LIN {X 0,Y 541.517,Z 483.658,A -85,B 0,C 180,E1 4032.092,E2 4032.092} C_VEL
LIN {X 0,Y 540.4,Z 508.601,A -85,B 0,C 180,E1 4034.781,E2 4034.781} C_VEL
LIN {X 0,Y 539.621,Z 531.792,A -85,B 0,C 180,E1 4038.266,E2 4038.266} C_VEL
LIN {X 0,Y 539.263,Z 546.74,A -85,B 0,C 180,E1 4041.527,E2 4041.527} C_VEL
LIN {X 0,Y 539.076,Z 557.16,A -85,B 0,C 180,E1 4045.169,E2 4045.169} C_VEL
LIN {X 0,Y 538.968,Z 561.446,A -85,B 0,C 180,E1 4048.393,E2 4048.393} C_VEL
LIN {X 0,Y 538.979,Z 561.385,A -85,B 0,C 180,E1 4051.612,E2 4051.612} C_VEL
LIN {X 0,Y 539.098,Z 556.976,A -85,B 0,C 180,E1 4054.835,E2 4054.835} C_VEL
LIN {X 0,Y 539.274,Z 546.384,A -85,B 0,C 180,E1 4058.478,E2 4058.478} C_VEL
LIN {X 0,Y 539.639,Z 530.084,A -85,B 0,C 180,E1 4061.943,E2 4061.943} C_VEL
LIN {X 0,Y 540.473,Z 506.897,A -85,B 0,C 180,E1 4065.337,E2 4065.337} C_VEL
LIN {X 0,Y 541.656,Z 481.261,A -85,B 0,C 180,E1 4068.039,E2 4068.039} C_VEL
LIN {X 0,Y 543.03,Z 451.784,A -85,B 0,C 180,E1 4070.227,E2 4070.227} C_VEL
LIN {X 0,Y 544.237,Z 421.039,A -85,B 0,C 180,E1 4071.776,E2 4071.776} C_VEL
LIN {X 0,Y 544.348,Z 387.144,A -85,B 0,C 180,E1 4072.819,E2 4072.819} C_VEL
LIN {X 0,Y 538.422,Z 370.16,A -85,B 0,C 180,E1 4073.523,E2 4073.523} C_VEL
LIN {X 0,Y 538.216,Z 370.16,A -85,B 0,C 180,E1 4079.313,E2 4079.313} C_VEL
LIN {X 0,Y 538.135,Z 370.16,A -85,B 0,C 180,E1 4085.331,E2 4085.331} C_VEL
LIN {X 0,Y 538.098,Z 370.16,A -85,B 0,C 180,E1 4090.57,E2 4090.57} C_VEL
LIN {X 0,Y 538.199,Z 370.16,A -85,B 0,C 180,E1 4097.005,E2 4097.005} C_VEL
LIN {X 0,Y 538.211,Z 370.16,A -85,B 0,C 180,E1 4101.967,E2 4101.967} C_VEL
LIN {X 0,Y 538.141,Z 370.16,A -85,B 0,C 180,E1 4107.691,E2 4107.691} C_VEL
LIN {X 0,Y 538.372,Z 370.16,A -85,B 0,C 180,E1 4113.263,E2 4113.263} C_VEL
LIN {X 0,Y 538.444,Z 370.16,A -85,B 0,C 180,E1 4118.562,E2 4118.562} C_VEL
LIN {X 0,Y 538.537,Z 370.16,A -85,B 0,C 180,E1 4123.674,E2 4123.674} C_VEL
LIN {X 0,Y 538.543,Z 370.16,A -85,B 0,C 180,E1 4128.652,E2 4128.652} C_VEL
LIN {X 0,Y 538.567,Z 370.16,A -85,B 0,C 180,E1 4133.545,E2 4133.545} C_VEL
LIN {X 0,Y 538.637,Z 370.16,A -85,B 0,C 180,E1 4138.39,E2 4138.39} C_VEL
LIN {X 0,Y 538.602,Z 370.16,A -85,B 0,C 180,E1 4143.224,E2 4143.224} C_VEL
LIN {X 0,Y 538.512,Z 370.16,A -85,B 0,C 180,E1 4148.082,E2 4148.082} C_VEL
LIN {X 0,Y 538.484,Z 370.16,A -85,B 0,C 180,E1 4152.999,E2 4152.999} C_VEL
LIN {X 0,Y 538.425,Z 370.16,A -85,B 0,C 180,E1 4158.018,E2 4158.018} C_VEL
LIN {X 0,Y 538.392,Z 370.16,A -85,B 0,C 180,E1 4163.184,E2 4163.184} C_VEL
LIN {X 0,Y 538.361,Z 370.16,A -85,B 0,C 180,E1 4165.152,E2 4165.152} C_VEL
LIN {X 0,Y 537.043,Z 370.16,A -85,B 0,C 180,E1 4166.074,E2 4166.074} C_VEL
LIN {X 0,Y 530.382,Z 370.16,A -85,B 0,C 180,E1 4168.584,E2 4168.584} C_VEL
LIN {X 0,Y 530.303,Z 370.16,A -85,B 0,C 180,E1 4168.822,E2 4168.822} C_VEL
LIN {X 0,Y 530.316,Z 370.16,A -85,B 0,C 180,E1 4174.817,E2 4174.817} C_VEL
LIN {X 0,Y 530.257,Z 370.16,A -85,B 0,C 180,E1 4181.047,E2 4181.047} C_VEL
LIN {X 0,Y 530.306,Z 370.16,A -85,B 0,C 180,E1 4186.749,E2 4186.749} C_VEL
LIN {X 0,Y 530.279,Z 370.16,A -85,B 0,C 180,E1 4193.16,E2 4193.16} C_VEL
LIN {X 0,Y 530.257,Z 370.16,A -85,B 0,C 180,E1 4199.072,E2 4199.072} C_VEL
LIN {X 0,Y 530.443,Z 370.823,A -85,B 0,C 180,E1 4200.434,E2 4200.434} C_VEL
LIN {X 0,Y 539.972,Z 394.145,A -85,B 0,C 180,E1 4201.321,E2 4201.321} C_VEL
LIN {X 0,Y 539.426,Z 441.23,A -85,B 0,C 180,E1 4202.159,E2 4202.159} C_VEL
LIN {X 0,Y 538.185,Z 477.288,A -85,B 0,C 180,E1 4203.418,E2 4203.418} C_VEL
LIN {X 0,Y 536.636,Z 511.971,A -85,B 0,C 180,E1 4205.296,E2 4205.296} C_VEL
LIN {X 0,Y 534.86,Z 545.508,A -85,B 0,C 180,E1 4207.882,E2 4207.882} C_VEL
LIN {X 0,Y 533.35,Z 574.49,A -85,B 0,C 180,E1 4210.945,E2 4210.945} C_VEL
LIN {X 0,Y 532.266,Z 598.279,A -85,B 0,C 180,E1 4214.321,E2 4214.321} C_VEL
LIN {X 0,Y 531.508,Z 617.476,A -85,B 0,C 180,E1 4218.08,E2 4218.08} C_VEL
LIN {X 0,Y 531.215,Z 630.601,A -85,B 0,C 180,E1 4221.805,E2 4221.805} C_VEL
LIN {X 0,Y 531.108,Z 637.962,A -85,B 0,C 180,E1 4225.092,E2 4225.092} C_VEL
LIN {X 0,Y 531.031,Z 641.508,A -85,B 0,C 180,E1 4228.364,E2 4228.364} C_VEL
LIN {X 0,Y 531.091,Z 641.512,A -85,B 0,C 180,E1 4231.631,E2 4231.631} C_VEL
LIN {X 0,Y 531.113,Z 637.97,A -85,B 0,C 180,E1 4234.903,E2 4234.903} C_VEL
LIN {X 0,Y 531.284,Z 628.183,A -85,B 0,C 180,E1 4239.014,E2 4239.014} C_VEL
LIN {X 0,Y 531.626,Z 613.791,A -85,B 0,C 180,E1 4242.748,E2 4242.748} C_VEL
LIN {X 0,Y 532.369,Z 594.338,A -85,B 0,C 180,E1 4246.307,E2 4246.307} C_VEL
LIN {X 0,Y 533.592,Z 569.267,A -85,B 0,C 180,E1 4249.687,E2 4249.687} C_VEL
LIN {X 0,Y 535.172,Z 539.83,A -85,B 0,C 180,E1 4252.617,E2 4252.617} C_VEL
LIN {X 0,Y 536.928,Z 506.945,A -85,B 0,C 180,E1 4255.018,E2 4255.018} C_VEL
LIN {X 0,Y 538.474,Z 472.313,A -85,B 0,C 180,E1 4256.797,E2 4256.797} C_VEL
LIN {X 0,Y 539.646,Z 435.196,A -85,B 0,C 180,E1 4257.986,E2 4257.986} C_VEL
LIN {X 0,Y 539.599,Z 392.517,A -85,B 0,C 180,E1 4258.725,E2 4258.725} C_VEL
LIN {X 0,Y 530.512,Z 370.16,A -85,B 0,C 180,E1 4259.603,E2 4259.603} C_VEL
LIN {X 0,Y 530.417,Z 370.16,A -85,B 0,C 180,E1 4264.806,E2 4264.806} C_VEL
LIN {X 0,Y 530.215,Z 370.16,A -85,B 0,C 180,E1 4271.047,E2 4271.047} C_VEL
LIN {X 0,Y 530.123,Z 370.16,A -85,B 0,C 180,E1 4276.733,E2 4276.733} C_VEL
LIN {X 0,Y 530.197,Z 370.16,A -85,B 0,C 180,E1 4283.155,E2 4283.155} C_VEL
LIN {X 0,Y 530.295,Z 370.16,A -85,B 0,C 180,E1 4289.077,E2 4289.077} C_VEL
LIN {X 0,Y 530.5,Z 370.16,A -85,B 0,C 180,E1 4294.654,E2 4294.654} C_VEL
LIN {X 0,Y 530.61,Z 370.872,A -85,B 0,C 180,E1 4296.73,E2 4296.73} C_VEL
LIN {X 0,Y 536.183,Z 392.946,A -85,B 0,C 180,E1 4297.301,E2 4297.301} C_VEL
LIN {X 0,Y 535.619,Z 427.462,A -85,B 0,C 180,E1 4298.388,E2 4298.388} C_VEL
LIN {X 0,Y 534.637,Z 459.023,A -85,B 0,C 180,E1 4300.06,E2 4300.06} C_VEL
LIN {X 0,Y 533.537,Z 487.309,A -85,B 0,C 180,E1 4302.269,E2 4302.269} C_VEL
LIN {X 0,Y 532.555,Z 511.968,A -85,B 0,C 180,E1 4304.986,E2 4304.986} C_VEL
LIN {X 0,Y 531.776,Z 531.931,A -85,B 0,C 180,E1 4308.087,E2 4308.087} C_VEL
LIN {X 0,Y 531.321,Z 548.213,A -85,B 0,C 180,E1 4311.808,E2 4311.808} C_VEL
LIN {X 0,Y 531.198,Z 557.105,A -85,B 0,C 180,E1 4315.094,E2 4315.094} C_VEL
LIN {X 0,Y 531.08,Z 561.45,A -85,B 0,C 180,E1 4318.365,E2 4318.365} C_VEL
LIN {X 0,Y 531.044,Z 561.418,A -85,B 0,C 180,E1 4321.633,E2 4321.633} C_VEL
LIN {X 0,Y 531.185,Z 556.932,A -85,B 0,C 180,E1 4324.904,E2 4324.904} C_VEL
LIN {X 0,Y 531.399,Z 546.438,A -85,B 0,C 180,E1 4328.601,E2 4328.601} C_VEL
LIN {X 0,Y 531.839,Z 529.134,A -85,B 0,C 180,E1 4332.326,E2 4332.326} C_VEL
LIN {X 0,Y 532.702,Z 507.725,A -85,B 0,C 180,E1 4335.45,E2 4335.45} C_VEL
LIN {X 0,Y 533.755,Z 482.611,A -85,B 0,C 180,E1 4338.067,E2 4338.067} C_VEL
LIN {X 0,Y 534.91,Z 453.057,A -85,B 0,C 180,E1 4340.248,E2 4340.248} C_VEL
LIN {X 0,Y 535.928,Z 420.413,A -85,B 0,C 180,E1 4341.854,E2 4341.854} C_VEL
LIN {X 0,Y 535.687,Z 387.806,A -85,B 0,C 180,E1 4342.835,E2 4342.835} C_VEL
LIN {X 0,Y 530.468,Z 370.16,A -85,B 0,C 180,E1 4343.4,E2 4343.4} C_VEL
LIN {X 0,Y 530.383,Z 370.16,A -85,B 0,C 180,E1 4349.027,E2 4349.027} C_VEL
LIN {X 0,Y 530.341,Z 370.16,A -85,B 0,C 180,E1 4354.813,E2 4354.813} C_VEL
LIN {X 0,Y 530.263,Z 370.16,A -85,B 0,C 180,E1 4361.044,E2 4361.044} C_VEL
LIN {X 0,Y 530.33,Z 370.16,A -85,B 0,C 180,E1 4366.758,E2 4366.758} C_VEL
LIN {X 0,Y 530.275,Z 370.16,A -85,B 0,C 180,E1 4373.166,E2 4373.166} C_VEL
LIN {X 0,Y 530.286,Z 370.16,A -85,B 0,C 180,E1 4379.08,E2 4379.08} C_VEL
LIN {X 0,Y 530.494,Z 370.16,A -85,B 0,C 180,E1 4384.657,E2 4384.657} C_VEL
LIN {X 0,Y 530.579,Z 370.16,A -85,B 0,C 180,E1 4385.986,E2 4385.986} C_VEL
LIN {X 0,Y 537.911,Z 392.099,A -85,B 0,C 180,E1 4386.837,E2 4386.837} C_VEL
LIN {X 0,Y 537.063,Z 426.025,A -85,B 0,C 180,E1 4387.945,E2 4387.945} C_VEL
LIN {X 0,Y 535.666,Z 456.498,A -85,B 0,C 180,E1 4389.59,E2 4389.59} C_VEL
LIN {X 0,Y 534.104,Z 484.887,A -85,B 0,C 180,E1 4391.835,E2 4391.835} C_VEL
LIN {X 0,Y 532.815,Z 509.576,A -85,B 0,C 180,E1 4394.554,E2 4394.554} C_VEL
LIN {X 0,Y 531.861,Z 529.926,A -85,B 0,C 180,E1 4397.676,E2 4397.676} C_VEL
LIN {X 0,Y 531.395,Z 546.737,A -85,B 0,C 180,E1 4401.4,E2 4401.4} C_VEL
LIN {X 0,Y 531.186,Z 557.158,A -85,B 0,C 180,E1 4405.098,E2 4405.098} C_VEL
LIN {X 0,Y 531.065,Z 561.445,A -85,B 0,C 180,E1 4408.369,E2 4408.369} C_VEL
LIN {X 0,Y 531.076,Z 561.385,A -85,B 0,C 180,E1 4411.636,E2 4411.636} C_VEL
LIN {X 0,Y 531.207,Z 556.977,A -85,B 0,C 180,E1 4414.907,E2 4414.907} C_VEL
LIN {X 0,Y 531.404,Z 546.387,A -85,B 0,C 180,E1 4418.604,E2 4418.604} C_VEL
LIN {X 0,Y 531.909,Z 529.402,A -85,B 0,C 180,E1 4422.328,E2 4422.328} C_VEL
LIN {X 0,Y 532.871,Z 509.001,A -85,B 0,C 180,E1 4425.428,E2 4425.428} C_VEL
LIN {X 0,Y 534.174,Z 483.9,A -85,B 0,C 180,E1 4428.168,E2 4428.168} C_VEL
LIN {X 0,Y 535.714,Z 454.866,A -85,B 0,C 180,E1 4430.426,E2 4430.426} C_VEL
LIN {X 0,Y 537.128,Z 423.446,A -85,B 0,C 180,E1 4432.08,E2 4432.08} C_VEL
LIN {X 0,Y 537.394,Z 389.167,A -85,B 0,C 180,E1 4433.17,E2 4433.17} C_VEL
LIN {X 0,Y 530.53,Z 370.16,A -85,B 0,C 180,E1 4433.979,E2 4433.979} C_VEL
LIN {X 0,Y 530.324,Z 370.16,A -85,B 0,C 180,E1 4439.035,E2 4439.035} C_VEL
LIN {X 0,Y 530.253,Z 370.16,A -85,B 0,C 180,E1 4444.824,E2 4444.824} C_VEL
LIN {X 0,Y 530.155,Z 370.16,A -85,B 0,C 180,E1 4451.059,E2 4451.059} C_VEL
LIN {X 0,Y 530.295,Z 370.16,A -85,B 0,C 180,E1 4456.753,E2 4456.753} C_VEL
LIN {X 0,Y 530.218,Z 370.16,A -85,B 0,C 180,E1 4463.085,E2 4463.085} C_VEL
LIN {X 0,Y 530.24,Z 370.16,A -85,B 0,C 180,E1 4469.076,E2 4469.076} C_VEL
LIN {X 0,Y 530.498,Z 370.16,A -85,B 0,C 180,E1 4474.657,E2 4474.657} C_VEL
LIN {X 0,Y 530.632,Z 370.16,A -85,B 0,C 180,E1 4480.314,E2 4480.314} C_VEL
LIN {X 0,Y 530.693,Z 370.16,A -85,B 0,C 180,E1 4485.924,E2 4485.924} C_VEL
LIN {X 0,Y 530.722,Z 370.16,A -85,B 0,C 180,E1 4491.801,E2 4491.801} C_VEL
LIN {X 0,Y 530.88,Z 370.16,A -85,B 0,C 180,E1 4496.732,E2 4496.732} C_VEL
LIN {X 0,Y 530.952,Z 370.16,A -85,B 0,C 180,E1 4501.635,E2 4501.635} C_VEL
LIN {X 0,Y 530.841,Z 370.16,A -85,B 0,C 180,E1 4506.551,E2 4506.551} C_VEL
LIN {X 0,Y 530.652,Z 370.16,A -85,B 0,C 180,E1 4511.521,E2 4511.521} C_VEL
LIN {X 0,Y 530.549,Z 370.16,A -85,B 0,C 180,E1 4516.581,E2 4516.581} C_VEL
LIN {X 0,Y 530.524,Z 370.16,A -85,B 0,C 180,E1 4521.777,E2 4521.777} C_VEL
LIN {X 0,Y 530.327,Z 370.16,A -85,B 0,C 180,E1 4527.748,E2 4527.748} C_VEL
LIN {X 0,Y 530.303,Z 370.16,A -85,B 0,C 180,E1 4528.822,E2 4528.822} C_VEL
LIN {X 0,Y 527.774,Z 370.16,A -85,B 0,C 180,E1 4530.211,E2 4530.211} C_VEL
LIN {X 0,Y 522.404,Z 370.16,A -85,B 0,C 180,E1 4532.292,E2 4532.292} C_VEL
LIN {X 0,Y 522.331,Z 370.16,A -85,B 0,C 180,E1 4532.533,E2 4532.533} C_VEL
LIN {X 0,Y 522.368,Z 370.16,A -85,B 0,C 180,E1 4538.505,E2 4538.505} C_VEL
LIN {X 0,Y 522.34,Z 370.16,A -85,B 0,C 180,E1 4544.076,E2 4544.076} C_VEL
LIN {X 0,Y 522.375,Z 370.16,A -85,B 0,C 180,E1 4550.384,E2 4550.384} C_VEL
LIN {X 0,Y 522.337,Z 370.16,A -85,B 0,C 180,E1 4556.583,E2 4556.583} C_VEL
LIN {X 0,Y 522.483,Z 370.16,A -85,B 0,C 180,E1 4559.982,E2 4559.982} C_VEL
LIN {X 0,Y 533.184,Z 398.599,A -85,B 0,C 180,E1 4560.988,E2 4560.988} C_VEL
LIN {X 0,Y 532.347,Z 444.004,A -85,B 0,C 180,E1 4561.837,E2 4561.837} C_VEL
LIN {X 0,Y 530.986,Z 479.733,A -85,B 0,C 180,E1 4563.144,E2 4563.144} C_VEL
LIN {X 0,Y 529.159,Z 515.25,A -85,B 0,C 180,E1 4565.149,E2 4565.149} C_VEL
LIN {X 0,Y 527.308,Z 546.909,A -85,B 0,C 180,E1 4567.684,E2 4567.684} C_VEL
LIN {X 0,Y 525.751,Z 574.49,A -85,B 0,C 180,E1 4570.659,E2 4570.659} C_VEL
LIN {X 0,Y 524.481,Z 598.279,A -85,B 0,C 180,E1 4574.082,E2 4574.082} C_VEL
LIN {X 0,Y 523.667,Z 617.477,A -85,B 0,C 180,E1 4577.899,E2 4577.899} C_VEL
LIN {X 0,Y 523.335,Z 630.601,A -85,B 0,C 180,E1 4581.681,E2 4581.681} C_VEL
LIN {X 0,Y 523.213,Z 637.961,A -85,B 0,C 180,E1 4585.018,E2 4585.018} C_VEL
LIN {X 0,Y 523.146,Z 641.509,A -85,B 0,C 180,E1 4588.339,E2 4588.339} C_VEL
LIN {X 0,Y 523.202,Z 641.512,A -85,B 0,C 180,E1 4591.656,E2 4591.656} C_VEL
LIN {X 0,Y 523.207,Z 637.97,A -85,B 0,C 180,E1 4594.977,E2 4594.977} C_VEL
LIN {X 0,Y 523.387,Z 629.464,A -85,B 0,C 180,E1 4598.732,E2 4598.732} C_VEL
LIN {X 0,Y 523.756,Z 615.735,A -85,B 0,C 180,E1 4602.518,E2 4602.518} C_VEL
LIN {X 0,Y 524.554,Z 595.663,A -85,B 0,C 180,E1 4606.341,E2 4606.341} C_VEL
LIN {X 0,Y 525.905,Z 571.028,A -85,B 0,C 180,E1 4609.768,E2 4609.768} C_VEL
LIN {X 0,Y 527.674,Z 541.222,A -85,B 0,C 180,E1 4612.834,E2 4612.834} C_VEL
LIN {X 0,Y 529.587,Z 508.646,A -85,B 0,C 180,E1 4615.276,E2 4615.276} C_VEL
LIN {X 0,Y 531.303,Z 473.736,A -85,B 0,C 180,E1 4617.121,E2 4617.121} C_VEL
LIN {X 0,Y 532.619,Z 437.259,A -85,B 0,C 180,E1 4618.34,E2 4618.34} C_VEL
LIN {X 0,Y 532.484,Z 394.319,A -85,B 0,C 180,E1 4619.117,E2 4619.117} C_VEL
LIN {X 0,Y 522.573,Z 370.16,A -85,B 0,C 180,E1 4620.064,E2 4620.064} C_VEL
LIN {X 0,Y 522.407,Z 370.16,A -85,B 0,C 180,E1 4625.763,E2 4625.763} C_VEL
LIN {X 0,Y 522.275,Z 370.16,A -85,B 0,C 180,E1 4631.81,E2 4631.81} C_VEL
LIN {X 0,Y 522.231,Z 370.16,A -85,B 0,C 180,E1 4638.182,E2 4638.182} C_VEL
LIN {X 0,Y 522.261,Z 370.16,A -85,B 0,C 180,E1 4644.566,E2 4644.566} C_VEL
LIN {X 0,Y 522.4,Z 370.16,A -85,B 0,C 180,E1 4650.483,E2 4650.483} C_VEL
LIN {X 0,Y 522.638,Z 370.16,A -85,B 0,C 180,E1 4656.388,E2 4656.388} C_VEL
LIN {X 0,Y 528.676,Z 392.668,A -85,B 0,C 180,E1 4657.022,E2 4657.022} C_VEL
LIN {X 0,Y 528.103,Z 427.602,A -85,B 0,C 180,E1 4658.119,E2 4658.119} C_VEL
LIN {X 0,Y 527.054,Z 459.805,A -85,B 0,C 180,E1 4659.836,E2 4659.836} C_VEL
LIN {X 0,Y 525.853,Z 488.687,A -85,B 0,C 180,E1 4662.127,E2 4662.127} C_VEL
LIN {X 0,Y 524.81,Z 513.709,A -85,B 0,C 180,E1 4664.951,E2 4664.951} C_VEL
LIN {X 0,Y 523.97,Z 533.559,A -85,B 0,C 180,E1 4668.119,E2 4668.119} C_VEL
LIN {X 0,Y 523.494,Z 548.685,A -85,B 0,C 180,E1 4671.685,E2 4671.685} C_VEL
LIN {X 0,Y 523.3,Z 557.335,A -85,B 0,C 180,E1 4675.02,E2 4675.02} C_VEL
LIN {X 0,Y 523.192,Z 561.543,A -85,B 0,C 180,E1 4678.341,E2 4678.341} C_VEL
LIN {X 0,Y 523.157,Z 561.506,A -85,B 0,C 180,E1 4681.657,E2 4681.657} C_VEL
LIN {X 0,Y 523.292,Z 557.138,A -85,B 0,C 180,E1 4684.978,E2 4684.978} C_VEL
LIN {X 0,Y 523.55,Z 546.828,A -85,B 0,C 180,E1 4688.731,E2 4688.731} C_VEL
LIN {X 0,Y 524.017,Z 530.672,A -85,B 0,C 180,E1 4692.301,E2 4692.301} C_VEL
LIN {X 0,Y 524.957,Z 509.65,A -85,B 0,C 180,E1 4695.47,E2 4695.47} C_VEL
LIN {X 0,Y 526.07,Z 484.343,A -85,B 0,C 180,E1 4698.188,E2 4698.188} C_VEL
LIN {X 0,Y 527.33,Z 454.86,A -85,B 0,C 180,E1 4700.42,E2 4700.42} C_VEL
LIN {X 0,Y 528.401,Z 423.505,A -85,B 0,C 180,E1 4702.028,E2 4702.028} C_VEL
LIN {X 0,Y 528.546,Z 390.358,A -85,B 0,C 180,E1 4703.074,E2 4703.074} C_VEL
LIN {X 0,Y 522.542,Z 370.16,A -85,B 0,C 180,E1 4703.69,E2 4703.69} C_VEL
LIN {X 0,Y 522.406,Z 370.16,A -85,B 0,C 180,E1 4709.616,E2 4709.616} C_VEL
LIN {X 0,Y 522.391,Z 370.16,A -85,B 0,C 180,E1 4715.765,E2 4715.765} C_VEL
LIN {X 0,Y 522.352,Z 370.16,A -85,B 0,C 180,E1 4721.803,E2 4721.803} C_VEL
LIN {X 0,Y 522.397,Z 370.16,A -85,B 0,C 180,E1 4728.202,E2 4728.202} C_VEL
LIN {X 0,Y 522.309,Z 370.16,A -85,B 0,C 180,E1 4734.573,E2 4734.573} C_VEL
LIN {X 0,Y 522.392,Z 370.16,A -85,B 0,C 180,E1 4740.486,E2 4740.486} C_VEL
LIN {X 0,Y 522.624,Z 370.16,A -85,B 0,C 180,E1 4745.523,E2 4745.523} C_VEL
LIN {X 0,Y 530.956,Z 394.225,A -85,B 0,C 180,E1 4746.475,E2 4746.475} C_VEL
LIN {X 0,Y 529.995,Z 427.507,A -85,B 0,C 180,E1 4747.602,E2 4747.602} C_VEL
LIN {X 0,Y 528.398,Z 458.785,A -85,B 0,C 180,E1 4749.337,E2 4749.337} C_VEL
LIN {X 0,Y 526.663,Z 487.353,A -85,B 0,C 180,E1 4751.682,E2 4751.682} C_VEL
LIN {X 0,Y 525.148,Z 512.132,A -85,B 0,C 180,E1 4754.537,E2 4754.537} C_VEL
LIN {X 0,Y 524.103,Z 533.026,A -85,B 0,C 180,E1 4757.914,E2 4757.914} C_VEL
LIN {X 0,Y 523.566,Z 547.353,A -85,B 0,C 180,E1 4761.271,E2 4761.271} C_VEL
LIN {X 0,Y 523.287,Z 557.383,A -85,B 0,C 180,E1 4765.023,E2 4765.023} C_VEL
LIN {X 0,Y 523.177,Z 561.528,A -85,B 0,C 180,E1 4768.344,E2 4768.344} C_VEL
LIN {X 0,Y 523.189,Z 561.47,A -85,B 0,C 180,E1 4771.661,E2 4771.661} C_VEL
LIN {X 0,Y 523.314,Z 557.211,A -85,B 0,C 180,E1 4774.981,E2 4774.981} C_VEL
LIN {X 0,Y 523.595,Z 547.027,A -85,B 0,C 180,E1 4778.734,E2 4778.734} C_VEL
LIN {X 0,Y 524.163,Z 531.432,A -85,B 0,C 180,E1 4782.301,E2 4782.301} C_VEL
LIN {X 0,Y 525.324,Z 509.902,A -85,B 0,C 180,E1 4785.677,E2 4785.677} C_VEL
LIN {X 0,Y 526.847,Z 484.366,A -85,B 0,C 180,E1 4788.515,E2 4788.515} C_VEL
LIN {X 0,Y 528.525,Z 455.971,A -85,B 0,C 180,E1 4790.756,E2 4790.756} C_VEL
LIN {X 0,Y 530.049,Z 424.907,A -85,B 0,C 180,E1 4792.428,E2 4792.428} C_VEL
LIN {X 0,Y 530.453,Z 391.054,A -85,B 0,C 180,E1 4793.537,E2 4793.537} C_VEL
LIN {X 0,Y 522.561,Z 370.16,A -85,B 0,C 180,E1 4794.425,E2 4794.425} C_VEL
LIN {X 0,Y 522.352,Z 370.16,A -85,B 0,C 180,E1 4799.605,E2 4799.605} C_VEL
LIN {X 0,Y 522.262,Z 370.16,A -85,B 0,C 180,E1 4805.437,E2 4805.437} C_VEL
LIN {X 0,Y 522.266,Z 370.16,A -85,B 0,C 180,E1 4811.818,E2 4811.818} C_VEL
LIN {X 0,Y 522.371,Z 370.16,A -85,B 0,C 180,E1 4818.198,E2 4818.198} C_VEL
LIN {X 0,Y 522.257,Z 370.16,A -85,B 0,C 180,E1 4824.568,E2 4824.568} C_VEL
LIN {X 0,Y 522.346,Z 370.16,A -85,B 0,C 180,E1 4830.483,E2 4830.483} C_VEL
LIN {X 0,Y 522.562,Z 370.16,A -85,B 0,C 180,E1 4836.073,E2 4836.073} C_VEL
LIN {X 0,Y 522.659,Z 370.16,A -85,B 0,C 180,E1 4841.422,E2 4841.422} C_VEL
LIN {X 0,Y 522.788,Z 370.16,A -85,B 0,C 180,E1 4846.606,E2 4846.606} C_VEL
LIN {X 0,Y 522.805,Z 370.16,A -85,B 0,C 180,E1 4851.676,E2 4851.676} C_VEL
LIN {X 0,Y 522.996,Z 370.16,A -85,B 0,C 180,E1 4856.682,E2 4856.682} C_VEL
LIN {X 0,Y 523.043,Z 370.16,A -85,B 0,C 180,E1 4861.66,E2 4861.66} C_VEL
LIN {X 0,Y 522.914,Z 370.16,A -85,B 0,C 180,E1 4866.651,E2 4866.651} C_VEL
LIN {X 0,Y 522.72,Z 370.16,A -85,B 0,C 180,E1 4871.698,E2 4871.698} C_VEL
LIN {X 0,Y 522.588,Z 370.16,A -85,B 0,C 180,E1 4877.05,E2 4877.05} C_VEL
LIN {X 0,Y 522.582,Z 370.16,A -85,B 0,C 180,E1 4882.125,E2 4882.125} C_VEL
LIN {X 0,Y 522.433,Z 370.16,A -85,B 0,C 180,E1 4887.624,E2 4887.624} C_VEL
LIN {X 0,Y 522.331,Z 370.16,A -85,B 0,C 180,E1 4892.533,E2 4892.533} C_VEL
LIN {X 0,Y 519.892,Z 370.16,A -85,B 0,C 180,E1 4893.947,E2 4893.947} C_VEL
LIN {X 0,Y 514.441,Z 370.16,A -85,B 0,C 180,E1 4896.312,E2 4896.312} C_VEL
LIN {X 0,Y 514.383,Z 370.16,A -85,B 0,C 180,E1 4902.605,E2 4902.605} C_VEL
LIN {X 0,Y 514.431,Z 370.16,A -85,B 0,C 180,E1 4907.397,E2 4907.397} C_VEL
LIN {X 0,Y 514.432,Z 370.16,A -85,B 0,C 180,E1 4912.617,E2 4912.617} C_VEL
LIN {X 0,Y 514.483,Z 370.16,A -85,B 0,C 180,E1 4919.323,E2 4919.323} C_VEL
LIN {X 0,Y 514.574,Z 371.189,A -85,B 0,C 180,E1 4919.611,E2 4919.611} C_VEL
LIN {X 0,Y 526.051,Z 399.878,A -85,B 0,C 180,E1 4920.641,E2 4920.641} C_VEL
LIN {X 0,Y 525.303,Z 442.719,A -85,B 0,C 180,E1 4921.425,E2 4921.425} C_VEL
LIN {X 0,Y 523.963,Z 478.034,A -85,B 0,C 180,E1 4922.674,E2 4922.674} C_VEL
LIN {X 0,Y 522.036,Z 513.663,A -85,B 0,C 180,E1 4924.672,E2 4924.672} C_VEL
LIN {X 0,Y 519.96,Z 545.628,A -85,B 0,C 180,E1 4927.225,E2 4927.225} C_VEL
LIN {X 0,Y 518.146,Z 574.489,A -85,B 0,C 180,E1 4930.363,E2 4930.363} C_VEL
LIN {X 0,Y 516.714,Z 598.279,A -85,B 0,C 180,E1 4933.836,E2 4933.836} C_VEL
LIN {X 0,Y 515.861,Z 617.477,A -85,B 0,C 180,E1 4937.713,E2 4937.713} C_VEL
LIN {X 0,Y 515.484,Z 630.601,A -85,B 0,C 180,E1 4941.553,E2 4941.553} C_VEL
LIN {X 0,Y 515.307,Z 639.168,A -85,B 0,C 180,E1 4945.785,E2 4945.785} C_VEL
LIN {X 0,Y 515.23,Z 642,A -85,B 0,C 180,E1 4949.997,E2 4949.997} C_VEL
LIN {X 0,Y 515.306,Z 639.176,A -85,B 0,C 180,E1 4954.21,E2 4954.21} C_VEL
LIN {X 0,Y 515.507,Z 630.612,A -85,B 0,C 180,E1 4958.441,E2 4958.441} C_VEL
LIN {X 0,Y 515.869,Z 617.498,A -85,B 0,C 180,E1 4962.282,E2 4962.282} C_VEL
LIN {X 0,Y 516.692,Z 598.309,A -85,B 0,C 180,E1 4966.159,E2 4966.159} C_VEL
LIN {X 0,Y 518.109,Z 574.532,A -85,B 0,C 180,E1 4969.633,E2 4969.633} C_VEL
LIN {X 0,Y 519.99,Z 545.732,A -85,B 0,C 180,E1 4972.763,E2 4972.763} C_VEL
LIN {X 0,Y 522.081,Z 513.747,A -85,B 0,C 180,E1 4975.32,E2 4975.32} C_VEL
LIN {X 0,Y 523.948,Z 479.224,A -85,B 0,C 180,E1 4977.27,E2 4977.27} C_VEL
LIN {X 0,Y 525.254,Z 443.124,A -85,B 0,C 180,E1 4978.566,E2 4978.566} C_VEL
LIN {X 0,Y 525.802,Z 397.642,A -85,B 0,C 180,E1 4979.404,E2 4979.404} C_VEL
LIN {X 0,Y 514.618,Z 370.16,A -85,B 0,C 180,E1 4980.483,E2 4980.483} C_VEL
LIN {X 0,Y 514.484,Z 370.16,A -85,B 0,C 180,E1 4986.049,E2 4986.049} C_VEL
LIN {X 0,Y 514.407,Z 370.16,A -85,B 0,C 180,E1 4990.348,E2 4990.348} C_VEL
LIN {X 0,Y 514.277,Z 370.16,A -85,B 0,C 180,E1 4997.384,E2 4997.384} C_VEL
LIN {X 0,Y 514.315,Z 370.16,A -85,B 0,C 180,E1 5002.629,E2 5002.629} C_VEL
LIN {X 0,Y 514.461,Z 370.16,A -85,B 0,C 180,E1 5008.578,E2 5008.578} C_VEL
LIN {X 0,Y 514.598,Z 370.16,A -85,B 0,C 180,E1 5013.813,E2 5013.813} C_VEL
LIN {X 0,Y 514.733,Z 370.824,A -85,B 0,C 180,E1 5016.122,E2 5016.122} C_VEL
LIN {X 0,Y 521.211,Z 395.938,A -85,B 0,C 180,E1 5016.818,E2 5016.818} C_VEL
LIN {X 0,Y 520.538,Z 429.526,A -85,B 0,C 180,E1 5017.92,E2 5017.92} C_VEL
LIN {X 0,Y 519.452,Z 461.076,A -85,B 0,C 180,E1 5019.639,E2 5019.639} C_VEL
LIN {X 0,Y 518.297,Z 488.419,A -85,B 0,C 180,E1 5021.826,E2 5021.826} C_VEL
LIN {X 0,Y 517.167,Z 512.469,A -85,B 0,C 180,E1 5024.506,E2 5024.506} C_VEL
LIN {X 0,Y 516.229,Z 532.942,A -85,B 0,C 180,E1 5027.723,E2 5027.723} C_VEL
LIN {X 0,Y 515.731,Z 547.793,A -85,B 0,C 180,E1 5031.134,E2 5031.134} C_VEL
LIN {X 0,Y 515.438,Z 558.027,A -85,B 0,C 180,E1 5034.944,E2 5034.944} C_VEL
LIN {X 0,Y 515.342,Z 562.207,A -85,B 0,C 180,E1 5038.315,E2 5038.315} C_VEL
LIN {X 0,Y 515.282,Z 562.133,A -85,B 0,C 180,E1 5041.682,E2 5041.682} C_VEL
LIN {X 0,Y 515.428,Z 557.764,A -85,B 0,C 180,E1 5045.054,E2 5045.054} C_VEL
LIN {X 0,Y 515.717,Z 547.31,A -85,B 0,C 180,E1 5048.864,E2 5048.864} C_VEL
LIN {X 0,Y 516.199,Z 532.212,A -85,B 0,C 180,E1 5052.275,E2 5052.275} C_VEL
LIN {X 0,Y 517.209,Z 511.572,A -85,B 0,C 180,E1 5055.49,E2 5055.49} C_VEL
LIN {X 0,Y 518.344,Z 487.185,A -85,B 0,C 180,E1 5058.198,E2 5058.198} C_VEL
LIN {X 0,Y 519.63,Z 458.763,A -85,B 0,C 180,E1 5060.462,E2 5060.462} C_VEL
LIN {X 0,Y 520.862,Z 426.768,A -85,B 0,C 180,E1 5062.199,E2 5062.199} C_VEL
LIN {X 0,Y 521.224,Z 392.36,A -85,B 0,C 180,E1 5063.332,E2 5063.332} C_VEL
LIN {X 0,Y 514.663,Z 370.16,A -85,B 0,C 180,E1 5064.051,E2 5064.051} C_VEL
LIN {X 0,Y 514.468,Z 370.16,A -85,B 0,C 180,E1 5070.015,E2 5070.015} C_VEL
LIN {X 0,Y 514.483,Z 370.16,A -85,B 0,C 180,E1 5076.05,E2 5076.05} C_VEL
LIN {X 0,Y 514.475,Z 370.16,A -85,B 0,C 180,E1 5080.343,E2 5080.343} C_VEL
LIN {X 0,Y 514.421,Z 370.16,A -85,B 0,C 180,E1 5085.068,E2 5085.068} C_VEL
LIN {X 0,Y 514.468,Z 370.16,A -85,B 0,C 180,E1 5089.914,E2 5089.914} C_VEL
LIN {X 0,Y 514.37,Z 370.16,A -85,B 0,C 180,E1 5096.001,E2 5096.001} C_VEL
LIN {X 0,Y 514.538,Z 370.16,A -85,B 0,C 180,E1 5101.965,E2 5101.965} C_VEL
LIN {X 0,Y 514.741,Z 370.967,A -85,B 0,C 180,E1 5105.063,E2 5105.063} C_VEL
LIN {X 0,Y 524.047,Z 395.473,A -85,B 0,C 180,E1 5106.083,E2 5106.083} C_VEL
LIN {X 0,Y 522.992,Z 428.211,A -85,B 0,C 180,E1 5107.209,E2 5107.209} C_VEL
LIN {X 0,Y 521.302,Z 459.03,A -85,B 0,C 180,E1 5108.937,E2 5108.937} C_VEL
LIN {X 0,Y 519.333,Z 487.533,A -85,B 0,C 180,E1 5111.299,E2 5111.299} C_VEL
LIN {X 0,Y 517.579,Z 513.203,A -85,B 0,C 180,E1 5114.305,E2 5114.305} C_VEL
LIN {X 0,Y 516.404,Z 533.889,A -85,B 0,C 180,E1 5117.731,E2 5117.731} C_VEL
LIN {X 0,Y 515.751,Z 548.105,A -85,B 0,C 180,E1 5121.137,E2 5121.137} C_VEL
LIN {X 0,Y 515.424,Z 558.056,A -85,B 0,C 180,E1 5124.947,E2 5124.947} C_VEL
LIN {X 0,Y 515.302,Z 562.168,A -85,B 0,C 180,E1 5128.319,E2 5128.319} C_VEL
LIN {X 0,Y 515.314,Z 562.113,A -85,B 0,C 180,E1 5131.686,E2 5131.686} C_VEL
LIN {X 0,Y 515.455,Z 557.888,A -85,B 0,C 180,E1 5135.058,E2 5135.058} C_VEL
LIN {X 0,Y 515.771,Z 547.779,A -85,B 0,C 180,E1 5138.867,E2 5138.867} C_VEL
LIN {X 0,Y 516.464,Z 532.339,A -85,B 0,C 180,E1 5142.488,E2 5142.488} C_VEL
LIN {X 0,Y 517.773,Z 511.002,A -85,B 0,C 180,E1 5145.912,E2 5145.912} C_VEL
LIN {X 0,Y 519.487,Z 485.709,A -85,B 0,C 180,E1 5148.787,E2 5148.787} C_VEL
LIN {X 0,Y 521.365,Z 457.53,A -85,B 0,C 180,E1 5151.072,E2 5151.072} C_VEL
LIN {X 0,Y 523.059,Z 425.743,A -85,B 0,C 180,E1 5152.816,E2 5152.816} C_VEL
LIN {X 0,Y 523.469,Z 392.925,A -85,B 0,C 180,E1 5153.921,E2 5153.921} C_VEL
LIN {X 0,Y 514.65,Z 370.16,A -85,B 0,C 180,E1 5154.903,E2 5154.903} C_VEL
LIN {X 0,Y 514.439,Z 370.16,A -85,B 0,C 180,E1 5161.417,E2 5161.417} C_VEL
LIN {X 0,Y 514.308,Z 370.16,A -85,B 0,C 180,E1 5167.369,E2 5167.369} C_VEL
LIN {X 0,Y 514.344,Z 370.16,A -85,B 0,C 180,E1 5172.623,E2 5172.623} C_VEL
LIN {X 0,Y 514.42,Z 370.16,A -85,B 0,C 180,E1 5177.402,E2 5177.402} C_VEL
LIN {X 0,Y 514.354,Z 370.16,A -85,B 0,C 180,E1 5182.632,E2 5182.632} C_VEL
LIN {X 0,Y 514.395,Z 370.16,A -85,B 0,C 180,E1 5188.6,E2 5188.6} C_VEL
LIN {X 0,Y 514.585,Z 370.16,A -85,B 0,C 180,E1 5193.814,E2 5193.814} C_VEL
LIN {X 0,Y 514.684,Z 370.16,A -85,B 0,C 180,E1 5200.274,E2 5200.274} C_VEL
LIN {X 0,Y 514.859,Z 370.16,A -85,B 0,C 180,E1 5206.396,E2 5206.396} C_VEL
LIN {X 0,Y 514.917,Z 370.16,A -85,B 0,C 180,E1 5211.548,E2 5211.548} C_VEL
LIN {X 0,Y 515.084,Z 370.16,A -85,B 0,C 180,E1 5216.631,E2 5216.631} C_VEL
LIN {X 0,Y 515.065,Z 370.16,A -85,B 0,C 180,E1 5221.977,E2 5221.977} C_VEL
LIN {X 0,Y 515.002,Z 370.16,A -85,B 0,C 180,E1 5226.754,E2 5226.754} C_VEL
LIN {X 0,Y 514.791,Z 370.16,A -85,B 0,C 180,E1 5231.881,E2 5231.881} C_VEL
LIN {X 0,Y 514.692,Z 370.16,A -85,B 0,C 180,E1 5237.107,E2 5237.107} C_VEL
LIN {X 0,Y 514.635,Z 370.16,A -85,B 0,C 180,E1 5242.485,E2 5242.485} C_VEL
LIN {X 0,Y 514.483,Z 370.16,A -85,B 0,C 180,E1 5248.088,E2 5248.088} C_VEL
LIN {X 0,Y 514.397,Z 370.16,A -85,B 0,C 180,E1 5254.001,E2 5254.001} C_VEL
LIN {X 0,Y 514.441,Z 370.16,A -85,B 0,C 180,E1 5256.312,E2 5256.312} C_VEL
LIN {X 0,Y 511.86,Z 370.16,A -85,B 0,C 180,E1 5257.748,E2 5257.748} C_VEL
LIN {X 0,Y 506.469,Z 370.16,A -85,B 0,C 180,E1 5259.899,E2 5259.899} C_VEL
LIN {X 0,Y 506.374,Z 370.16,A -85,B 0,C 180,E1 5260.148,E2 5260.148} C_VEL
LIN {X 0,Y 506.451,Z 370.16,A -85,B 0,C 180,E1 5266.561,E2 5266.561} C_VEL
LIN {X 0,Y 506.502,Z 370.16,A -85,B 0,C 180,E1 5273.285,E2 5273.285} C_VEL
LIN {X 0,Y 506.583,Z 370.16,A -85,B 0,C 180,E1 5279.147,E2 5279.147} C_VEL
LIN {X 0,Y 518.649,Z 400.482,A -85,B 0,C 180,E1 5280.275,E2 5280.275} C_VEL
LIN {X 0,Y 518.019,Z 443.674,A -85,B 0,C 180,E1 5281.105,E2 5281.105} C_VEL
LIN {X 0,Y 516.497,Z 481.641,A -85,B 0,C 180,E1 5282.503,E2 5282.503} C_VEL
LIN {X 0,Y 514.559,Z 516.707,A -85,B 0,C 180,E1 5284.511,E2 5284.511} C_VEL
LIN {X 0,Y 512.399,Z 547.78,A -85,B 0,C 180,E1 5287.085,E2 5287.085} C_VEL
LIN {X 0,Y 510.422,Z 576.241,A -85,B 0,C 180,E1 5290.28,E2 5290.28} C_VEL
LIN {X 0,Y 508.845,Z 600.708,A -85,B 0,C 180,E1 5294.023,E2 5294.023} C_VEL
LIN {X 0,Y 507.939,Z 619.212,A -85,B 0,C 180,E1 5297.955,E2 5297.955} C_VEL
LIN {X 0,Y 507.571,Z 631.748,A -85,B 0,C 180,E1 5301.852,E2 5301.852} C_VEL
LIN {X 0,Y 507.406,Z 639.168,A -85,B 0,C 180,E1 5305.72,E2 5305.72} C_VEL
LIN {X 0,Y 507.343,Z 642,A -85,B 0,C 180,E1 5309.997,E2 5309.997} C_VEL
LIN {X 0,Y 507.403,Z 639.177,A -85,B 0,C 180,E1 5314.275,E2 5314.275} C_VEL
LIN {X 0,Y 507.613,Z 630.612,A -85,B 0,C 180,E1 5318.573,E2 5318.573} C_VEL
LIN {X 0,Y 508.023,Z 617.497,A -85,B 0,C 180,E1 5322.475,E2 5322.475} C_VEL
LIN {X 0,Y 508.955,Z 598.308,A -85,B 0,C 180,E1 5326.412,E2 5326.412} C_VEL
LIN {X 0,Y 510.497,Z 574.531,A -85,B 0,C 180,E1 5329.938,E2 5329.938} C_VEL
LIN {X 0,Y 512.525,Z 546.194,A -85,B 0,C 180,E1 5333.067,E2 5333.067} C_VEL
LIN {X 0,Y 514.711,Z 515.22,A -85,B 0,C 180,E1 5335.592,E2 5335.592} C_VEL
LIN {X 0,Y 516.622,Z 479.251,A -85,B 0,C 180,E1 5337.602,E2 5337.602} C_VEL
LIN {X 0,Y 518.041,Z 442.022,A -85,B 0,C 180,E1 5338.942,E2 5338.942} C_VEL
LIN {X 0,Y 518.365,Z 399.255,A -85,B 0,C 180,E1 5339.758,E2 5339.758} C_VEL
LIN {X 0,Y 506.689,Z 370.16,A -85,B 0,C 180,E1 5340.896,E2 5340.896} C_VEL
LIN {X 0,Y 506.549,Z 370.16,A -85,B 0,C 180,E1 5346.705,E2 5346.705} C_VEL
LIN {X 0,Y 506.309,Z 370.16,A -85,B 0,C 180,E1 5353.447,E2 5353.447} C_VEL
LIN {X 0,Y 506.304,Z 370.16,A -85,B 0,C 180,E1 5358.864,E2 5358.864} C_VEL
LIN {X 0,Y 506.431,Z 370.16,A -85,B 0,C 180,E1 5365.389,E2 5365.389} C_VEL
LIN {X 0,Y 506.545,Z 370.16,A -85,B 0,C 180,E1 5371.431,E2 5371.431} C_VEL
LIN {X 0,Y 506.793,Z 370.16,A -85,B 0,C 180,E1 5375.754,E2 5375.754} C_VEL
LIN {X 0,Y 513.763,Z 396.829,A -85,B 0,C 180,E1 5376.55,E2 5376.55} C_VEL
LIN {X 0,Y 512.999,Z 431.625,A -85,B 0,C 180,E1 5377.723,E2 5377.723} C_VEL
LIN {X 0,Y 511.817,Z 463.961,A -85,B 0,C 180,E1 5379.548,E2 5379.548} C_VEL
LIN {X 0,Y 510.466,Z 492.559,A -85,B 0,C 180,E1 5381.94,E2 5381.94} C_VEL
LIN {X 0,Y 509.307,Z 516.883,A -85,B 0,C 180,E1 5384.835,E2 5384.835} C_VEL
LIN {X 0,Y 508.355,Z 536.694,A -85,B 0,C 180,E1 5388.185,E2 5388.185} C_VEL
LIN {X 0,Y 507.775,Z 551.234,A -85,B 0,C 180,E1 5391.857,E2 5391.857} C_VEL
LIN {X 0,Y 507.541,Z 560.167,A -85,B 0,C 180,E1 5395.722,E2 5395.722} C_VEL
LIN {X 0,Y 507.477,Z 562.852,A -85,B 0,C 180,E1 5398.289,E2 5398.289} C_VEL
LIN {X 0,Y 507.42,Z 562.754,A -85,B 0,C 180,E1 5401.709,E2 5401.709} C_VEL
LIN {X 0,Y 507.582,Z 558.365,A -85,B 0,C 180,E1 5405.132,E2 5405.132} C_VEL
LIN {X 0,Y 507.829,Z 549.297,A -85,B 0,C 180,E1 5408.571,E2 5408.571} C_VEL
LIN {X 0,Y 508.382,Z 533.773,A -85,B 0,C 180,E1 5412.249,E2 5412.249} C_VEL
LIN {X 0,Y 509.452,Z 513.399,A -85,B 0,C 180,E1 5415.511,E2 5415.511} C_VEL
LIN {X 0,Y 510.629,Z 489.308,A -85,B 0,C 180,E1 5418.281,E2 5418.281} C_VEL
LIN {X 0,Y 512.085,Z 460.222,A -85,B 0,C 180,E1 5420.665,E2 5420.665} C_VEL
LIN {X 0,Y 513.42,Z 427.291,A -85,B 0,C 180,E1 5422.487,E2 5422.487} C_VEL
LIN {X 0,Y 513.741,Z 393.846,A -85,B 0,C 180,E1 5423.617,E2 5423.617} C_VEL
LIN {X 0,Y 506.693,Z 370.16,A -85,B 0,C 180,E1 5424.43,E2 5424.43} C_VEL
LIN {X 0,Y 506.541,Z 370.16,A -85,B 0,C 180,E1 5430.535,E2 5430.535} C_VEL
LIN {X 0,Y 506.581,Z 370.16,A -85,B 0,C 180,E1 5436.704,E2 5436.704} C_VEL
LIN {X 0,Y 506.465,Z 370.16,A -85,B 0,C 180,E1 5441.647,E2 5441.647} C_VEL
LIN {X 0,Y 506.483,Z 370.16,A -85,B 0,C 180,E1 5448.352,E2 5448.352} C_VEL
LIN {X 0,Y 506.506,Z 370.16,A -85,B 0,C 180,E1 5453.803,E2 5453.803} C_VEL
LIN {X 0,Y 506.537,Z 370.16,A -85,B 0,C 180,E1 5460.079,E2 5460.079} C_VEL
LIN {X 0,Y 506.783,Z 370.16,A -85,B 0,C 180,E1 5464.544,E2 5464.544} C_VEL
LIN {X 0,Y 517.105,Z 397.052,A -85,B 0,C 180,E1 5465.691,E2 5465.691} C_VEL
LIN {X 0,Y 516.001,Z 429.608,A -85,B 0,C 180,E1 5466.839,E2 5466.839} C_VEL
LIN {X 0,Y 514.214,Z 459.669,A -85,B 0,C 180,E1 5468.552,E2 5468.552} C_VEL
LIN {X 0,Y 512.108,Z 487.833,A -85,B 0,C 180,E1 5470.914,E2 5470.914} C_VEL
LIN {X 0,Y 510.167,Z 512.766,A -85,B 0,C 180,E1 5473.85,E2 5473.85} C_VEL
LIN {X 0,Y 508.749,Z 533.746,A -85,B 0,C 180,E1 5477.325,E2 5477.325} C_VEL
LIN {X 0,Y 507.953,Z 548.875,A -85,B 0,C 180,E1 5481,E2 5481} C_VEL
LIN {X 0,Y 507.573,Z 558.73,A -85,B 0,C 180,E1 5484.869,E2 5484.869} C_VEL
LIN {X 0,Y 507.44,Z 562.809,A -85,B 0,C 180,E1 5488.293,E2 5488.293} C_VEL
LIN {X 0,Y 507.45,Z 562.753,A -85,B 0,C 180,E1 5491.712,E2 5491.712} C_VEL
LIN {X 0,Y 507.609,Z 558.564,A -85,B 0,C 180,E1 5495.136,E2 5495.136} C_VEL
LIN {X 0,Y 507.969,Z 548.563,A -85,B 0,C 180,E1 5499.005,E2 5499.005} C_VEL
LIN {X 0,Y 508.783,Z 533.262,A -85,B 0,C 180,E1 5502.679,E2 5502.679} C_VEL
LIN {X 0,Y 510.249,Z 512.109,A -85,B 0,C 180,E1 5506.153,E2 5506.153} C_VEL
LIN {X 0,Y 512.163,Z 486.908,A -85,B 0,C 180,E1 5509.09,E2 5509.09} C_VEL
LIN {X 0,Y 514.3,Z 458.137,A -85,B 0,C 180,E1 5511.46,E2 5511.46} C_VEL
LIN {X 0,Y 516.056,Z 426.993,A -85,B 0,C 180,E1 5513.195,E2 5513.195} C_VEL
LIN {X 0,Y 516.582,Z 395.408,A -85,B 0,C 180,E1 5514.29,E2 5514.29} C_VEL
LIN {X 0,Y 506.687,Z 370.16,A -85,B 0,C 180,E1 5515.423,E2 5515.423} C_VEL
LIN {X 0,Y 506.497,Z 370.16,A -85,B 0,C 180,E1 5520.543,E2 5520.543} C_VEL
LIN {X 0,Y 506.418,Z 370.16,A -85,B 0,C 180,E1 5526.723,E2 5526.723} C_VEL
LIN {X 0,Y 506.389,Z 370.16,A -85,B 0,C 180,E1 5533.446,E2 5533.446} C_VEL
LIN {X 0,Y 506.44,Z 370.16,A -85,B 0,C 180,E1 5538.881,E2 5538.881} C_VEL
LIN {X 0,Y 506.419,Z 370.16,A -85,B 0,C 180,E1 5545.391,E2 5545.391} C_VEL
LIN {X 0,Y 506.509,Z 370.16,A -85,B 0,C 180,E1 5551.432,E2 5551.432} C_VEL
LIN {X 0,Y 506.718,Z 370.16,A -85,B 0,C 180,E1 5557.146,E2 5557.146} C_VEL
LIN {X 0,Y 506.859,Z 370.16,A -85,B 0,C 180,E1 5562.911,E2 5562.911} C_VEL
LIN {X 0,Y 506.888,Z 370.16,A -85,B 0,C 180,E1 5567.933,E2 5567.933} C_VEL
LIN {X 0,Y 506.945,Z 370.16,A -85,B 0,C 180,E1 5573.141,E2 5573.141} C_VEL
LIN {X 0,Y 507.044,Z 370.16,A -85,B 0,C 180,E1 5578.29,E2 5578.29} C_VEL
LIN {X 0,Y 507.031,Z 370.16,A -85,B 0,C 180,E1 5583.425,E2 5583.425} C_VEL
LIN {X 0,Y 506.903,Z 370.16,A -85,B 0,C 180,E1 5588.589,E2 5588.589} C_VEL
LIN {X 0,Y 506.834,Z 370.16,A -85,B 0,C 180,E1 5593.826,E2 5593.826} C_VEL
LIN {X 0,Y 506.738,Z 370.16,A -85,B 0,C 180,E1 5599.187,E2 5599.187} C_VEL
LIN {X 0,Y 506.662,Z 370.16,A -85,B 0,C 180,E1 5604.73,E2 5604.73} C_VEL
LIN {X 0,Y 506.5,Z 370.16,A -85,B 0,C 180,E1 5610.54,E2 5610.54} C_VEL
LIN {X 0,Y 506.552,Z 370.16,A -85,B 0,C 180,E1 5616.709,E2 5616.709} C_VEL
LIN {X 0,Y 506.374,Z 370.16,A -85,B 0,C 180,E1 5620.148,E2 5620.148} C_VEL
LIN {X 0,Y 505.117,Z 370.16,A -85,B 0,C 180,E1 5621.127,E2 5621.127} C_VEL
LIN {X 0,Y 498.585,Z 370.16,A -85,B 0,C 180,E1 5623.797,E2 5623.797} C_VEL
LIN {X 0,Y 498.504,Z 370.16,A -85,B 0,C 180,E1 5624.05,E2 5624.05} C_VEL
LIN {X 0,Y 498.501,Z 370.16,A -85,B 0,C 180,E1 5630.371,E2 5630.371} C_VEL
LIN {X 0,Y 498.511,Z 370.16,A -85,B 0,C 180,E1 5636.86,E2 5636.86} C_VEL
LIN {X 0,Y 498.695,Z 370.54,A -85,B 0,C 180,E1 5638.729,E2 5638.729} C_VEL
LIN {X 0,Y 511.614,Z 403.073,A -85,B 0,C 180,E1 5639.945,E2 5639.945} C_VEL
LIN {X 0,Y 510.804,Z 443.533,A -85,B 0,C 180,E1 5640.746,E2 5640.746} C_VEL
LIN {X 0,Y 509.12,Z 481.969,A -85,B 0,C 180,E1 5642.191,E2 5642.191} C_VEL
LIN {X 0,Y 507.046,Z 516.807,A -85,B 0,C 180,E1 5644.224,E2 5644.224} C_VEL
LIN {X 0,Y 504.92,Z 548.187,A -85,B 0,C 180,E1 5646.778,E2 5646.778} C_VEL
LIN {X 0,Y 502.827,Z 576.241,A -85,B 0,C 180,E1 5649.969,E2 5649.969} C_VEL
LIN {X 0,Y 501.076,Z 600.707,A -85,B 0,C 180,E1 5653.768,E2 5653.768} C_VEL
LIN {X 0,Y 500.099,Z 619.212,A -85,B 0,C 180,E1 5657.763,E2 5657.763} C_VEL
LIN {X 0,Y 499.684,Z 631.748,A -85,B 0,C 180,E1 5661.723,E2 5661.723} C_VEL
LIN {X 0,Y 499.525,Z 639.169,A -85,B 0,C 180,E1 5665.652,E2 5665.652} C_VEL
LIN {X 0,Y 499.446,Z 642,A -85,B 0,C 180,E1 5669.997,E2 5669.997} C_VEL
LIN {X 0,Y 499.521,Z 639.177,A -85,B 0,C 180,E1 5674.343,E2 5674.343} C_VEL
LIN {X 0,Y 499.737,Z 630.611,A -85,B 0,C 180,E1 5678.71,E2 5678.71} C_VEL
LIN {X 0,Y 500.184,Z 617.496,A -85,B 0,C 180,E1 5682.673,E2 5682.673} C_VEL
LIN {X 0,Y 501.205,Z 598.308,A -85,B 0,C 180,E1 5686.673,E2 5686.673} C_VEL
LIN {X 0,Y 502.896,Z 574.531,A -85,B 0,C 180,E1 5690.252,E2 5690.252} C_VEL
LIN {X 0,Y 505.03,Z 546.814,A -85,B 0,C 180,E1 5693.352,E2 5693.352} C_VEL
LIN {X 0,Y 507.324,Z 513.688,A -85,B 0,C 180,E1 5695.992,E2 5695.992} C_VEL
LIN {X 0,Y 509.328,Z 478.366,A -85,B 0,C 180,E1 5697.971,E2 5697.971} C_VEL
LIN {X 0,Y 510.836,Z 441.269,A -85,B 0,C 180,E1 5699.32,E2 5699.32} C_VEL
LIN {X 0,Y 511.282,Z 401.534,A -85,B 0,C 180,E1 5700.096,E2 5700.096} C_VEL
LIN {X 0,Y 498.752,Z 370.16,A -85,B 0,C 180,E1 5701.294,E2 5701.294} C_VEL
LIN {X 0,Y 498.539,Z 370.16,A -85,B 0,C 180,E1 5707.395,E2 5707.395} C_VEL
LIN {X 0,Y 498.389,Z 370.16,A -85,B 0,C 180,E1 5713.194,E2 5713.194} C_VEL
LIN {X 0,Y 498.345,Z 370.16,A -85,B 0,C 180,E1 5719.414,E2 5719.414} C_VEL
LIN {X 0,Y 498.514,Z 370.16,A -85,B 0,C 180,E1 5725.076,E2 5725.076} C_VEL
LIN {X 0,Y 498.623,Z 370.16,A -85,B 0,C 180,E1 5731.698,E2 5731.698} C_VEL
LIN {X 0,Y 498.862,Z 370.16,A -85,B 0,C 180,E1 5735.415,E2 5735.415} C_VEL
LIN {X 0,Y 506.325,Z 398.248,A -85,B 0,C 180,E1 5736.278,E2 5736.278} C_VEL
LIN {X 0,Y 505.511,Z 432.581,A -85,B 0,C 180,E1 5737.463,E2 5737.463} C_VEL
LIN {X 0,Y 504.315,Z 463.691,A -85,B 0,C 180,E1 5739.23,E2 5739.23} C_VEL
LIN {X 0,Y 502.917,Z 491.825,A -85,B 0,C 180,E1 5741.58,E2 5741.58} C_VEL
LIN {X 0,Y 501.652,Z 516.413,A -85,B 0,C 180,E1 5744.486,E2 5744.486} C_VEL
LIN {X 0,Y 500.641,Z 536.135,A -85,B 0,C 180,E1 5747.778,E2 5747.778} C_VEL
LIN {X 0,Y 500.033,Z 550.461,A -85,B 0,C 180,E1 5751.292,E2 5751.292} C_VEL
LIN {X 0,Y 499.735,Z 559.331,A -85,B 0,C 180,E1 5754.784,E2 5754.784} C_VEL
LIN {X 0,Y 499.623,Z 563.511,A -85,B 0,C 180,E1 5758.262,E2 5758.262} C_VEL
LIN {X 0,Y 499.565,Z 563.388,A -85,B 0,C 180,E1 5761.735,E2 5761.735} C_VEL
LIN {X 0,Y 499.733,Z 558.953,A -85,B 0,C 180,E1 5765.213,E2 5765.213} C_VEL
LIN {X 0,Y 500.077,Z 548.351,A -85,B 0,C 180,E1 5769.127,E2 5769.127} C_VEL
LIN {X 0,Y 500.631,Z 532.974,A -85,B 0,C 180,E1 5772.663,E2 5772.663} C_VEL
LIN {X 0,Y 501.825,Z 512.037,A -85,B 0,C 180,E1 5775.978,E2 5775.978} C_VEL
LIN {X 0,Y 503.271,Z 486.004,A -85,B 0,C 180,E1 5778.893,E2 5778.893} C_VEL
LIN {X 0,Y 504.784,Z 456.627,A -85,B 0,C 180,E1 5781.208,E2 5781.208} C_VEL
LIN {X 0,Y 506.192,Z 423.846,A -85,B 0,C 180,E1 5782.944,E2 5782.944} C_VEL
LIN {X 0,Y 506.289,Z 395.389,A -85,B 0,C 180,E1 5783.907,E2 5783.907} C_VEL
LIN {X 0,Y 498.759,Z 370.16,A -85,B 0,C 180,E1 5784.75,E2 5784.75} C_VEL
LIN {X 0,Y 498.567,Z 370.16,A -85,B 0,C 180,E1 5791.077,E2 5791.077} C_VEL
LIN {X 0,Y 498.594,Z 370.16,A -85,B 0,C 180,E1 5797.391,E2 5797.391} C_VEL
LIN {X 0,Y 498.543,Z 370.16,A -85,B 0,C 180,E1 5803.217,E2 5803.217} C_VEL
LIN {X 0,Y 498.502,Z 370.16,A -85,B 0,C 180,E1 5809.394,E2 5809.394} C_VEL
LIN {X 0,Y 498.54,Z 370.16,A -85,B 0,C 180,E1 5815.073,E2 5815.073} C_VEL
LIN {X 0,Y 498.616,Z 370.16,A -85,B 0,C 180,E1 5821.701,E2 5821.701} C_VEL
LIN {X 0,Y 498.822,Z 370.237,A -85,B 0,C 180,E1 5824.062,E2 5824.062} C_VEL
LIN {X 0,Y 510.138,Z 399.671,A -85,B 0,C 180,E1 5825.338,E2 5825.338} C_VEL
LIN {X 0,Y 508.819,Z 433.241,A -85,B 0,C 180,E1 5826.577,E2 5826.577} C_VEL
LIN {X 0,Y 506.769,Z 464.169,A -85,B 0,C 180,E1 5828.443,E2 5828.443} C_VEL
LIN {X 0,Y 504.601,Z 491.461,A -85,B 0,C 180,E1 5830.848,E2 5830.848} C_VEL
LIN {X 0,Y 502.507,Z 515.42,A -85,B 0,C 180,E1 5833.821,E2 5833.821} C_VEL
LIN {X 0,Y 500.998,Z 535.682,A -85,B 0,C 180,E1 5837.348,E2 5837.348} C_VEL
LIN {X 0,Y 500.084,Z 551.049,A -85,B 0,C 180,E1 5841.296,E2 5841.296} C_VEL
LIN {X 0,Y 499.723,Z 559.41,A -85,B 0,C 180,E1 5844.788,E2 5844.788} C_VEL
LIN {X 0,Y 499.576,Z 563.449,A -85,B 0,C 180,E1 5848.266,E2 5848.266} C_VEL
LIN {X 0,Y 499.582,Z 563.397,A -85,B 0,C 180,E1 5851.739,E2 5851.739} C_VEL
LIN {X 0,Y 499.757,Z 559.25,A -85,B 0,C 180,E1 5855.217,E2 5855.217} C_VEL
LIN {X 0,Y 500.159,Z 549.34,A -85,B 0,C 180,E1 5859.146,E2 5859.146} C_VEL
LIN {X 0,Y 501.082,Z 534.207,A -85,B 0,C 180,E1 5862.878,E2 5862.878} C_VEL
LIN {X 0,Y 502.736,Z 513.262,A -85,B 0,C 180,E1 5866.401,E2 5866.401} C_VEL
LIN {X 0,Y 504.826,Z 488.327,A -85,B 0,C 180,E1 5869.378,E2 5869.378} C_VEL
LIN {X 0,Y 507.073,Z 460.377,A -85,B 0,C 180,E1 5871.744,E2 5871.744} C_VEL
LIN {X 0,Y 509.002,Z 428.881,A -85,B 0,C 180,E1 5873.536,E2 5873.536} C_VEL
LIN {X 0,Y 509.415,Z 397.08,A -85,B 0,C 180,E1 5874.688,E2 5874.688} C_VEL
LIN {X 0,Y 498.747,Z 370.16,A -85,B 0,C 180,E1 5875.904,E2 5875.904} C_VEL
LIN {X 0,Y 498.523,Z 370.16,A -85,B 0,C 180,E1 5881.758,E2 5881.758} C_VEL
LIN {X 0,Y 498.408,Z 370.16,A -85,B 0,C 180,E1 5887.84,E2 5887.84} C_VEL
LIN {X 0,Y 498.497,Z 370.16,A -85,B 0,C 180,E1 5894.311,E2 5894.311} C_VEL
LIN {X 0,Y 498.467,Z 370.16,A -85,B 0,C 180,E1 5900.374,E2 5900.374} C_VEL
LIN {X 0,Y 498.487,Z 370.16,A -85,B 0,C 180,E1 5906.863,E2 5906.863} C_VEL
LIN {X 0,Y 498.643,Z 370.16,A -85,B 0,C 180,E1 5912.91,E2 5912.91} C_VEL
LIN {X 0,Y 498.836,Z 370.16,A -85,B 0,C 180,E1 5918.644,E2 5918.644} C_VEL
LIN {X 0,Y 498.965,Z 370.16,A -85,B 0,C 180,E1 5924.154,E2 5924.154} C_VEL
LIN {X 0,Y 499.047,Z 370.16,A -85,B 0,C 180,E1 5929.514,E2 5929.514} C_VEL
LIN {X 0,Y 499.138,Z 370.16,A -85,B 0,C 180,E1 5934.781,E2 5934.781} C_VEL
LIN {X 0,Y 499.259,Z 370.16,A -85,B 0,C 180,E1 5940.001,E2 5940.001} C_VEL
LIN {X 0,Y 499.163,Z 370.16,A -85,B 0,C 180,E1 5945.222,E2 5945.222} C_VEL
LIN {X 0,Y 499.001,Z 370.16,A -85,B 0,C 180,E1 5950.489,E2 5950.489} C_VEL
LIN {X 0,Y 498.887,Z 370.16,A -85,B 0,C 180,E1 5955.851,E2 5955.851} C_VEL
LIN {X 0,Y 498.803,Z 370.16,A -85,B 0,C 180,E1 5961.36,E2 5961.36} C_VEL
LIN {X 0,Y 498.635,Z 370.16,A -85,B 0,C 180,E1 5967.093,E2 5967.093} C_VEL
LIN {X 0,Y 498.537,Z 370.16,A -85,B 0,C 180,E1 5973.136,E2 5973.136} C_VEL
LIN {X 0,Y 498.513,Z 370.16,A -85,B 0,C 180,E1 5979.625,E2 5979.625} C_VEL
LIN {X 0,Y 498.504,Z 370.16,A -85,B 0,C 180,E1 5984.05,E2 5984.05} C_VEL
LIN {X 0,Y 496.072,Z 370.16,A -85,B 0,C 180,E1 5985.526,E2 5985.526} C_VEL
LIN {X 0,Y 490.612,Z 370.16,A -85,B 0,C 180,E1 5987.994,E2 5987.994} C_VEL
LIN {X 0,Y 490.556,Z 370.16,A -85,B 0,C 180,E1 5994.097,E2 5994.097} C_VEL
LIN {X 0,Y 490.726,Z 370.16,A -85,B 0,C 180,E1 5998.238,E2 5998.238} C_VEL
LIN {X 0,Y 504.532,Z 405.631,A -85,B 0,C 180,E1 5999.606,E2 5999.606} C_VEL
LIN {X 0,Y 503.46,Z 447.115,A -85,B 0,C 180,E1 6000.48,E2 6000.48} C_VEL
LIN {X 0,Y 501.613,Z 484.455,A -85,B 0,C 180,E1 6001.983,E2 6001.983} C_VEL
LIN {X 0,Y 499.351,Z 519.356,A -85,B 0,C 180,E1 6004.108,E2 6004.108} C_VEL
LIN {X 0,Y 497.006,Z 552.125,A -85,B 0,C 180,E1 6006.907,E2 6006.907} C_VEL
LIN {X 0,Y 494.95,Z 579.598,A -85,B 0,C 180,E1 6010.116,E2 6010.116} C_VEL
LIN {X 0,Y 493.259,Z 601.908,A -85,B 0,C 180,E1 6013.733,E2 6013.733} C_VEL
LIN {X 0,Y 492.289,Z 619.211,A -85,B 0,C 180,E1 6017.566,E2 6017.566} C_VEL
LIN {X 0,Y 491.815,Z 631.748,A -85,B 0,C 180,E1 6021.59,E2 6021.59} C_VEL
LIN {X 0,Y 491.642,Z 639.168,A -85,B 0,C 180,E1 6025.582,E2 6025.582} C_VEL
LIN {X 0,Y 491.547,Z 642,A -85,B 0,C 180,E1 6029.997,E2 6029.997} C_VEL
LIN {X 0,Y 491.637,Z 639.177,A -85,B 0,C 180,E1 6034.413,E2 6034.413} C_VEL
LIN {X 0,Y 491.847,Z 630.611,A -85,B 0,C 180,E1 6038.85,E2 6038.85} C_VEL
LIN {X 0,Y 492.362,Z 617.495,A -85,B 0,C 180,E1 6042.878,E2 6042.878} C_VEL
LIN {X 0,Y 493.471,Z 598.307,A -85,B 0,C 180,E1 6046.942,E2 6046.942} C_VEL
LIN {X 0,Y 495.279,Z 574.855,A -85,B 0,C 180,E1 6050.52,E2 6050.52} C_VEL
LIN {X 0,Y 497.434,Z 546.393,A -85,B 0,C 180,E1 6053.643,E2 6053.643} C_VEL
LIN {X 0,Y 499.853,Z 513.273,A -85,B 0,C 180,E1 6056.323,E2 6056.323} C_VEL
LIN {X 0,Y 502.029,Z 477.455,A -85,B 0,C 180,E1 6058.354,E2 6058.354} C_VEL
LIN {X 0,Y 503.689,Z 440.462,A -85,B 0,C 180,E1 6059.706,E2 6059.706} C_VEL
LIN {X 0,Y 503.776,Z 402.874,A -85,B 0,C 180,E1 6060.484,E2 6060.484} C_VEL
LIN {X 0,Y 490.864,Z 370.16,A -85,B 0,C 180,E1 6061.806,E2 6061.806} C_VEL
LIN {X 0,Y 490.583,Z 370.16,A -85,B 0,C 180,E1 6068.108,E2 6068.108} C_VEL
LIN {X 0,Y 490.455,Z 370.16,A -85,B 0,C 180,E1 6074.767,E2 6074.767} C_VEL
LIN {X 0,Y 490.452,Z 370.16,A -85,B 0,C 180,E1 6080.503,E2 6080.503} C_VEL
LIN {X 0,Y 490.622,Z 370.16,A -85,B 0,C 180,E1 6086.419,E2 6086.419} C_VEL
LIN {X 0,Y 490.721,Z 370.16,A -85,B 0,C 180,E1 6092.433,E2 6092.433} C_VEL
LIN {X 0,Y 490.893,Z 370.16,A -85,B 0,C 180,E1 6095.044,E2 6095.044} C_VEL
LIN {X 0,Y 498.911,Z 401.59,A -85,B 0,C 180,E1 6096.044,E2 6096.044} C_VEL
LIN {X 0,Y 497.988,Z 435.803,A -85,B 0,C 180,E1 6097.298,E2 6097.298} C_VEL
LIN {X 0,Y 496.709,Z 466.611,A -85,B 0,C 180,E1 6099.131,E2 6099.131} C_VEL
LIN {X 0,Y 495.206,Z 494.521,A -85,B 0,C 180,E1 6101.548,E2 6101.548} C_VEL
LIN {X 0,Y 493.917,Z 518.495,A -85,B 0,C 180,E1 6104.488,E2 6104.488} C_VEL
LIN {X 0,Y 492.813,Z 537.694,A -85,B 0,C 180,E1 6107.806,E2 6107.806} C_VEL
LIN {X 0,Y 492.151,Z 552.45,A -85,B 0,C 180,E1 6111.597,E2 6111.597} C_VEL
LIN {X 0,Y 491.83,Z 561.477,A -85,B 0,C 180,E1 6115.585,E2 6115.585} C_VEL
LIN {X 0,Y 491.774,Z 564.172,A -85,B 0,C 180,E1 6118.235,E2 6118.235} C_VEL
LIN {X 0,Y 491.691,Z 564.031,A -85,B 0,C 180,E1 6121.763,E2 6121.763} C_VEL
LIN {X 0,Y 491.885,Z 559.541,A -85,B 0,C 180,E1 6125.297,E2 6125.297} C_VEL
LIN {X 0,Y 492.243,Z 549.114,A -85,B 0,C 180,E1 6129.197,E2 6129.197} C_VEL
LIN {X 0,Y 492.858,Z 533.341,A -85,B 0,C 180,E1 6132.866,E2 6132.866} C_VEL
LIN {X 0,Y 494.147,Z 512.246,A -85,B 0,C 180,E1 6136.233,E2 6136.233} C_VEL
LIN {X 0,Y 495.695,Z 486.105,A -85,B 0,C 180,E1 6139.186,E2 6139.186} C_VEL
LIN {X 0,Y 497.346,Z 456.394,A -85,B 0,C 180,E1 6141.541,E2 6141.541} C_VEL
LIN {X 0,Y 498.775,Z 424.628,A -85,B 0,C 180,E1 6143.239,E2 6143.239} C_VEL
LIN {X 0,Y 498.819,Z 396.687,A -85,B 0,C 180,E1 6144.211,E2 6144.211} C_VEL
LIN {X 0,Y 490.834,Z 370.16,A -85,B 0,C 180,E1 6145.187,E2 6145.187} C_VEL
LIN {X 0,Y 490.681,Z 370.16,A -85,B 0,C 180,E1 6151.633,E2 6151.633} C_VEL
LIN {X 0,Y 490.655,Z 370.16,A -85,B 0,C 180,E1 6158.103,E2 6158.103} C_VEL
LIN {X 0,Y 490.617,Z 370.16,A -85,B 0,C 180,E1 6164.791,E2 6164.791} C_VEL
LIN {X 0,Y 490.59,Z 370.16,A -85,B 0,C 180,E1 6170.484,E2 6170.484} C_VEL
LIN {X 0,Y 490.622,Z 370.16,A -85,B 0,C 180,E1 6176.42,E2 6176.42} C_VEL
LIN {X 0,Y 490.894,Z 370.16,A -85,B 0,C 180,E1 6183.503,E2 6183.503} C_VEL
LIN {X 0,Y 503.151,Z 401.913,A -85,B 0,C 180,E1 6184.972,E2 6184.972} C_VEL
LIN {X 0,Y 501.746,Z 434.496,A -85,B 0,C 180,E1 6186.208,E2 6186.208} C_VEL
LIN {X 0,Y 499.556,Z 465.16,A -85,B 0,C 180,E1 6188.092,E2 6188.092} C_VEL
LIN {X 0,Y 497.2,Z 493.108,A -85,B 0,C 180,E1 6190.601,E2 6190.601} C_VEL
LIN {X 0,Y 494.988,Z 516.552,A -85,B 0,C 180,E1 6193.569,E2 6193.569} C_VEL
LIN {X 0,Y 493.311,Z 536.611,A -85,B 0,C 180,E1 6197.147,E2 6197.147} C_VEL
LIN {X 0,Y 492.346,Z 550.624,A -85,B 0,C 180,E1 6200.768,E2 6200.768} C_VEL
LIN {X 0,Y 491.875,Z 560.092,A -85,B 0,C 180,E1 6204.705,E2 6204.705} C_VEL
LIN {X 0,Y 491.702,Z 564.092,A -85,B 0,C 180,E1 6208.238,E2 6208.238} C_VEL
LIN {X 0,Y 491.709,Z 564.038,A -85,B 0,C 180,E1 6211.767,E2 6211.767} C_VEL
LIN {X 0,Y 491.912,Z 559.933,A -85,B 0,C 180,E1 6215.3,E2 6215.3} C_VEL
LIN {X 0,Y 492.363,Z 550.292,A -85,B 0,C 180,E1 6219.246,E2 6219.246} C_VEL
LIN {X 0,Y 493.407,Z 535.157,A -85,B 0,C 180,E1 6223.081,E2 6223.081} C_VEL
LIN {X 0,Y 495.23,Z 514.397,A -85,B 0,C 180,E1 6226.657,E2 6226.657} C_VEL
LIN {X 0,Y 497.487,Z 489.569,A -85,B 0,C 180,E1 6229.676,E2 6229.676} C_VEL
LIN {X 0,Y 499.92,Z 460.944,A -85,B 0,C 180,E1 6232.129,E2 6232.129} C_VEL
LIN {X 0,Y 501.939,Z 430.051,A -85,B 0,C 180,E1 6233.91,E2 6233.91} C_VEL
LIN {X 0,Y 502.4,Z 399.143,A -85,B 0,C 180,E1 6235.067,E2 6235.067} C_VEL
LIN {X 0,Y 490.846,Z 370.16,A -85,B 0,C 180,E1 6236.431,E2 6236.431} C_VEL
LIN {X 0,Y 490.644,Z 370.16,A -85,B 0,C 180,E1 6241.641,E2 6241.641} C_VEL
LIN {X 0,Y 490.478,Z 370.16,A -85,B 0,C 180,E1 6248.125,E2 6248.125} C_VEL
LIN {X 0,Y 490.586,Z 370.16,A -85,B 0,C 180,E1 6254.786,E2 6254.786} C_VEL
LIN {X 0,Y 490.551,Z 370.16,A -85,B 0,C 180,E1 6260.497,E2 6260.497} C_VEL
LIN {X 0,Y 490.549,Z 370.16,A -85,B 0,C 180,E1 6266.441,E2 6266.441} C_VEL
LIN {X 0,Y 490.697,Z 370.16,A -85,B 0,C 180,E1 6272.435,E2 6272.435} C_VEL
LIN {X 0,Y 490.88,Z 370.16,A -85,B 0,C 180,E1 6278.28,E2 6278.28} C_VEL
LIN {X 0,Y 491.022,Z 370.16,A -85,B 0,C 180,E1 6283.891,E2 6283.891} C_VEL
LIN {X 0,Y 491.144,Z 370.16,A -85,B 0,C 180,E1 6290.551,E2 6290.551} C_VEL
LIN {X 0,Y 491.371,Z 370.16,A -85,B 0,C 180,E1 6296.468,E2 6296.468} C_VEL
LIN {X 0,Y 491.473,Z 370.16,A -85,B 0,C 180,E1 6301.766,E2 6301.766} C_VEL
LIN {X 0,Y 491.226,Z 370.16,A -85,B 0,C 180,E1 6307.082,E2 6307.082} C_VEL
LIN {X 0,Y 491.021,Z 370.16,A -85,B 0,C 180,E1 6312.465,E2 6312.465} C_VEL
LIN {X 0,Y 490.916,Z 370.16,A -85,B 0,C 180,E1 6317.963,E2 6317.963} C_VEL
LIN {X 0,Y 490.833,Z 370.16,A -85,B 0,C 180,E1 6323.64,E2 6323.64} C_VEL
LIN {X 0,Y 490.598,Z 370.16,A -85,B 0,C 180,E1 6330.221,E2 6330.221} C_VEL
LIN {X 0,Y 490.593,Z 370.16,A -85,B 0,C 180,E1 6336.642,E2 6336.642} C_VEL
LIN {X 0,Y 490.587,Z 370.16,A -85,B 0,C 180,E1 6342.759,E2 6342.759} C_VEL
LIN {X 0,Y 490.612,Z 370.16,A -85,B 0,C 180,E1 6347.994,E2 6347.994} C_VEL
LIN {X 0,Y 486.6,Z 370.16,A -85,B 0,C 180,E1 6349.974,E2 6349.974} C_VEL
LIN {X 0,Y 482.622,Z 370.16,A -85,B 0,C 180,E1 6351.986,E2 6351.986} C_VEL
LIN {X 0,Y 482.751,Z 370.16,A -85,B 0,C 180,E1 6357.721,E2 6357.721} C_VEL
LIN {X 0,Y 497.334,Z 407.274,A -85,B 0,C 180,E1 6359.239,E2 6359.239} C_VEL
LIN {X 0,Y 496.179,Z 448.015,A -85,B 0,C 180,E1 6360.143,E2 6360.143} C_VEL
LIN {X 0,Y 494.196,Z 485.733,A -85,B 0,C 180,E1 6361.711,E2 6361.711} C_VEL
LIN {X 0,Y 491.758,Z 520.715,A -85,B 0,C 180,E1 6363.903,E2 6363.903} C_VEL
LIN {X 0,Y 489.287,Z 553.084,A -85,B 0,C 180,E1 6366.762,E2 6366.762} C_VEL
LIN {X 0,Y 487.151,Z 580.248,A -85,B 0,C 180,E1 6370.008,E2 6370.008} C_VEL
LIN {X 0,Y 485.532,Z 601.901,A -85,B 0,C 180,E1 6373.467,E2 6373.467} C_VEL
LIN {X 0,Y 484.457,Z 619.21,A -85,B 0,C 180,E1 6377.362,E2 6377.362} C_VEL
LIN {X 0,Y 483.949,Z 631.748,A -85,B 0,C 180,E1 6381.452,E2 6381.452} C_VEL
LIN {X 0,Y 483.759,Z 639.167,A -85,B 0,C 180,E1 6385.51,E2 6385.51} C_VEL
LIN {X 0,Y 483.661,Z 642,A -85,B 0,C 180,E1 6389.997,E2 6389.997} C_VEL
LIN {X 0,Y 483.752,Z 639.176,A -85,B 0,C 180,E1 6394.485,E2 6394.485} C_VEL
LIN {X 0,Y 483.975,Z 630.611,A -85,B 0,C 180,E1 6398.996,E2 6398.996} C_VEL
LIN {X 0,Y 484.538,Z 617.494,A -85,B 0,C 180,E1 6403.09,E2 6403.09} C_VEL
LIN {X 0,Y 485.678,Z 599.485,A -85,B 0,C 180,E1 6406.989,E2 6406.989} C_VEL
LIN {X 0,Y 487.515,Z 574.897,A -85,B 0,C 180,E1 6410.714,E2 6410.714} C_VEL
LIN {X 0,Y 489.769,Z 546.579,A -85,B 0,C 180,E1 6413.885,E2 6413.885} C_VEL
LIN {X 0,Y 492.302,Z 514.364,A -85,B 0,C 180,E1 6416.554,E2 6416.554} C_VEL
LIN {X 0,Y 494.624,Z 478.949,A -85,B 0,C 180,E1 6418.63,E2 6418.63} C_VEL
LIN {X 0,Y 496.406,Z 442.008,A -85,B 0,C 180,E1 6420.033,E2 6420.033} C_VEL
LIN {X 0,Y 496.834,Z 405.428,A -85,B 0,C 180,E1 6420.822,E2 6420.822} C_VEL
LIN {X 0,Y 482.889,Z 370.16,A -85,B 0,C 180,E1 6422.315,E2 6422.315} C_VEL
LIN {X 0,Y 482.634,Z 370.16,A -85,B 0,C 180,E1 6428.852,E2 6428.852} C_VEL
LIN {X 0,Y 482.494,Z 370.16,A -85,B 0,C 180,E1 6433.806,E2 6433.806} C_VEL
LIN {X 0,Y 482.508,Z 370.16,A -85,B 0,C 180,E1 6438.849,E2 6438.849} C_VEL
LIN {X 0,Y 482.568,Z 370.16,A -85,B 0,C 180,E1 6444.65,E2 6444.65} C_VEL
LIN {X 0,Y 482.738,Z 370.16,A -85,B 0,C 180,E1 6449.881,E2 6449.881} C_VEL
LIN {X 0,Y 482.97,Z 370.844,A -85,B 0,C 180,E1 6454.674,E2 6454.674} C_VEL
LIN {X 0,Y 491.57,Z 401.302,A -85,B 0,C 180,E1 6455.702,E2 6455.702} C_VEL
LIN {X 0,Y 490.588,Z 435.376,A -85,B 0,C 180,E1 6456.944,E2 6456.944} C_VEL
LIN {X 0,Y 489.246,Z 466.502,A -85,B 0,C 180,E1 6458.797,E2 6458.797} C_VEL
LIN {X 0,Y 487.626,Z 494.689,A -85,B 0,C 180,E1 6461.25,E2 6461.25} C_VEL
LIN {X 0,Y 486.224,Z 519.142,A -85,B 0,C 180,E1 6464.279,E2 6464.279} C_VEL
LIN {X 0,Y 485.051,Z 538.22,A -85,B 0,C 180,E1 6467.608,E2 6467.608} C_VEL
LIN {X 0,Y 484.334,Z 553.057,A -85,B 0,C 180,E1 6471.46,E2 6471.46} C_VEL
LIN {X 0,Y 483.99,Z 562.128,A -85,B 0,C 180,E1 6475.514,E2 6475.514} C_VEL
LIN {X 0,Y 483.912,Z 564.832,A -85,B 0,C 180,E1 6478.206,E2 6478.206} C_VEL
LIN {X 0,Y 483.821,Z 564.667,A -85,B 0,C 180,E1 6481.792,E2 6481.792} C_VEL
LIN {X 0,Y 484.041,Z 560.127,A -85,B 0,C 180,E1 6485.383,E2 6485.383} C_VEL
LIN {X 0,Y 484.366,Z 550.807,A -85,B 0,C 180,E1 6488.99,E2 6488.99} C_VEL
LIN {X 0,Y 484.996,Z 536.057,A -85,B 0,C 180,E1 6492.62,E2 6492.62} C_VEL
LIN {X 0,Y 486.311,Z 515.421,A -85,B 0,C 180,E1 6496.082,E2 6496.082} C_VEL
LIN {X 0,Y 487.896,Z 490.093,A -85,B 0,C 180,E1 6499.096,E2 6499.096} C_VEL
LIN {X 0,Y 489.579,Z 461.113,A -85,B 0,C 180,E1 6501.542,E2 6501.542} C_VEL
LIN {X 0,Y 491.196,Z 428.808,A -85,B 0,C 180,E1 6503.392,E2 6503.392} C_VEL
LIN {X 0,Y 491.352,Z 397.979,A -85,B 0,C 180,E1 6504.52,E2 6504.52} C_VEL
LIN {X 0,Y 482.901,Z 370.16,A -85,B 0,C 180,E1 6505.566,E2 6505.566} C_VEL
LIN {X 0,Y 482.739,Z 370.16,A -85,B 0,C 180,E1 6512.216,E2 6512.216} C_VEL
LIN {X 0,Y 482.74,Z 370.16,A -85,B 0,C 180,E1 6518.843,E2 6518.843} C_VEL
LIN {X 0,Y 482.648,Z 370.16,A -85,B 0,C 180,E1 6523.83,E2 6523.83} C_VEL
LIN {X 0,Y 482.671,Z 370.16,A -85,B 0,C 180,E1 6528.829,E2 6528.829} C_VEL
LIN {X 0,Y 482.615,Z 370.16,A -85,B 0,C 180,E1 6534.644,E2 6534.644} C_VEL
LIN {X 0,Y 482.728,Z 370.16,A -85,B 0,C 180,E1 6539.885,E2 6539.885} C_VEL
LIN {X 0,Y 482.922,Z 370.646,A -85,B 0,C 180,E1 6543.02,E2 6543.02} C_VEL
LIN {X 0,Y 496.142,Z 404.593,A -85,B 0,C 180,E1 6544.611,E2 6544.611} C_VEL
LIN {X 0,Y 494.516,Z 437.521,A -85,B 0,C 180,E1 6545.928,E2 6545.928} C_VEL
LIN {X 0,Y 492.187,Z 468.593,A -85,B 0,C 180,E1 6547.928,E2 6547.928} C_VEL
LIN {X 0,Y 489.664,Z 495.574,A -85,B 0,C 180,E1 6550.459,E2 6550.459} C_VEL
LIN {X 0,Y 487.323,Z 519.055,A -85,B 0,C 180,E1 6553.535,E2 6553.535} C_VEL
LIN {X 0,Y 485.569,Z 538.548,A -85,B 0,C 180,E1 6557.168,E2 6557.168} C_VEL
LIN {X 0,Y 484.497,Z 552.586,A -85,B 0,C 180,E1 6561.014,E2 6561.014} C_VEL
LIN {X 0,Y 484.033,Z 560.777,A -85,B 0,C 180,E1 6564.619,E2 6564.619} C_VEL
LIN {X 0,Y 483.83,Z 564.733,A -85,B 0,C 180,E1 6568.21,E2 6568.21} C_VEL
LIN {X 0,Y 483.837,Z 564.684,A -85,B 0,C 180,E1 6571.796,E2 6571.796} C_VEL
LIN {X 0,Y 484.068,Z 560.626,A -85,B 0,C 180,E1 6575.386,E2 6575.386} C_VEL
LIN {X 0,Y 484.58,Z 551.321,A -85,B 0,C 180,E1 6579.322,E2 6579.322} C_VEL
LIN {X 0,Y 485.74,Z 536.079,A -85,B 0,C 180,E1 6583.292,E2 6583.292} C_VEL
LIN {X 0,Y 487.711,Z 515.375,A -85,B 0,C 180,E1 6586.921,E2 6586.921} C_VEL
LIN {X 0,Y 490.13,Z 490.626,A -85,B 0,C 180,E1 6589.983,E2 6589.983} C_VEL
LIN {X 0,Y 492.643,Z 462.686,A -85,B 0,C 180,E1 6592.43,E2 6592.43} C_VEL
LIN {X 0,Y 494.848,Z 431.56,A -85,B 0,C 180,E1 6594.274,E2 6594.274} C_VEL
LIN {X 0,Y 495.544,Z 401.773,A -85,B 0,C 180,E1 6595.422,E2 6595.422} C_VEL
LIN {X 0,Y 482.853,Z 370.16,A -85,B 0,C 180,E1 6596.934,E2 6596.934} C_VEL
LIN {X 0,Y 482.685,Z 370.16,A -85,B 0,C 180,E1 6602.225,E2 6602.225} C_VEL
LIN {X 0,Y 482.551,Z 370.16,A -85,B 0,C 180,E1 6608.867,E2 6608.867} C_VEL
LIN {X 0,Y 482.59,Z 370.16,A -85,B 0,C 180,E1 6613.822,E2 6613.822} C_VEL
LIN {X 0,Y 482.64,Z 370.16,A -85,B 0,C 180,E1 6618.84,E2 6618.84} C_VEL
LIN {X 0,Y 482.567,Z 370.16,A -85,B 0,C 180,E1 6624.659,E2 6624.659} C_VEL
LIN {X 0,Y 482.681,Z 370.16,A -85,B 0,C 180,E1 6629.88,E2 6629.88} C_VEL
LIN {X 0,Y 482.876,Z 370.16,A -85,B 0,C 180,E1 6635.949,E2 6635.949} C_VEL
LIN {X 0,Y 483.025,Z 370.16,A -85,B 0,C 180,E1 6641.736,E2 6641.736} C_VEL
LIN {X 0,Y 483.145,Z 370.16,A -85,B 0,C 180,E1 6647.331,E2 6647.331} C_VEL
LIN {X 0,Y 483.227,Z 370.16,A -85,B 0,C 180,E1 6652.802,E2 6652.802} C_VEL
LIN {X 0,Y 483.372,Z 370.16,A -85,B 0,C 180,E1 6658.206,E2 6658.206} C_VEL
LIN {X 0,Y 483.323,Z 370.16,A -85,B 0,C 180,E1 6663.593,E2 6663.593} C_VEL
LIN {X 0,Y 483.181,Z 370.16,A -85,B 0,C 180,E1 6669.014,E2 6669.014} C_VEL
LIN {X 0,Y 483.072,Z 370.16,A -85,B 0,C 180,E1 6674.521,E2 6674.521} C_VEL
LIN {X 0,Y 482.956,Z 370.16,A -85,B 0,C 180,E1 6680.172,E2 6680.172} C_VEL
LIN {X 0,Y 482.848,Z 370.16,A -85,B 0,C 180,E1 6686.038,E2 6686.038} C_VEL
LIN {X 0,Y 482.698,Z 370.16,A -85,B 0,C 180,E1 6692.222,E2 6692.222} C_VEL
LIN {X 0,Y 482.67,Z 370.16,A -85,B 0,C 180,E1 6698.853,E2 6698.853} C_VEL
LIN {X 0,Y 482.621,Z 370.16,A -85,B 0,C 180,E1 6703.819,E2 6703.819} C_VEL
LIN {X 0,Y 482.66,Z 370.16,A -85,B 0,C 180,E1 6708.834,E2 6708.834} C_VEL
LIN {X 0,Y 482.622,Z 370.16,A -85,B 0,C 180,E1 6711.986,E2 6711.986} C_VEL
LIN {X 0,Y 478.629,Z 370.16,A -85,B 0,C 180,E1 6714.008,E2 6714.008} C_VEL
LIN {X 0,Y 474.711,Z 370.16,A -85,B 0,C 180,E1 6716.064,E2 6716.064} C_VEL
LIN {X 0,Y 474.846,Z 370.654,A -85,B 0,C 180,E1 6717.236,E2 6717.236} C_VEL
LIN {X 0,Y 490.25,Z 411.342,A -85,B 0,C 180,E1 6718.907,E2 6718.907} C_VEL
LIN {X 0,Y 488.808,Z 450.824,A -85,B 0,C 180,E1 6719.866,E2 6719.866} C_VEL
LIN {X 0,Y 486.673,Z 487.954,A -85,B 0,C 180,E1 6721.487,E2 6721.487} C_VEL
LIN {X 0,Y 483.999,Z 524.011,A -85,B 0,C 180,E1 6723.856,E2 6723.856} C_VEL
LIN {X 0,Y 481.45,Z 555.139,A -85,B 0,C 180,E1 6726.729,E2 6726.729} C_VEL
LIN {X 0,Y 479.213,Z 582.537,A -85,B 0,C 180,E1 6730.144,E2 6730.144} C_VEL
LIN {X 0,Y 477.44,Z 605.951,A -85,B 0,C 180,E1 6734.125,E2 6734.125} C_VEL
LIN {X 0,Y 476.434,Z 622.466,A -85,B 0,C 180,E1 6738.077,E2 6738.077} C_VEL
LIN {X 0,Y 476.041,Z 632.837,A -85,B 0,C 180,E1 6741.769,E2 6741.769} C_VEL
LIN {X 0,Y 475.817,Z 640.16,A -85,B 0,C 180,E1 6746.349,E2 6746.349} C_VEL
LIN {X 0,Y 475.761,Z 642,A -85,B 0,C 180,E1 6749.997,E2 6749.997} C_VEL
LIN {X 0,Y 475.851,Z 639.176,A -85,B 0,C 180,E1 6754.559,E2 6754.559} C_VEL
LIN {X 0,Y 476.091,Z 630.61,A -85,B 0,C 180,E1 6759.146,E2 6759.146} C_VEL
LIN {X 0,Y 476.728,Z 617.47,A -85,B 0,C 180,E1 6763.294,E2 6763.294} C_VEL
LIN {X 0,Y 477.944,Z 597.737,A -85,B 0,C 180,E1 6767.432,E2 6767.432} C_VEL
LIN {X 0,Y 479.884,Z 572.977,A -85,B 0,C 180,E1 6771.165,E2 6771.165} C_VEL
LIN {X 0,Y 482.351,Z 544.41,A -85,B 0,C 180,E1 6774.365,E2 6774.365} C_VEL
LIN {X 0,Y 485.021,Z 511.829,A -85,B 0,C 180,E1 6777.046,E2 6777.046} C_VEL
LIN {X 0,Y 487.444,Z 476.512,A -85,B 0,C 180,E1 6779.092,E2 6779.092} C_VEL
LIN {X 0,Y 489.425,Z 438.598,A -85,B 0,C 180,E1 6780.508,E2 6780.508} C_VEL
LIN {X 0,Y 489.713,Z 407.718,A -85,B 0,C 180,E1 6781.185,E2 6781.185} C_VEL
LIN {X 0,Y 474.948,Z 370.16,A -85,B 0,C 180,E1 6782.809,E2 6782.809} C_VEL
LIN {X 0,Y 474.627,Z 370.16,A -85,B 0,C 180,E1 6789.635,E2 6789.635} C_VEL
LIN {X 0,Y 474.492,Z 370.16,A -85,B 0,C 180,E1 6795.416,E2 6795.416} C_VEL
LIN {X 0,Y 474.542,Z 370.16,A -85,B 0,C 180,E1 6800.352,E2 6800.352} C_VEL
LIN {X 0,Y 474.67,Z 370.16,A -85,B 0,C 180,E1 6806.017,E2 6806.017} C_VEL
LIN {X 0,Y 474.825,Z 370.16,A -85,B 0,C 180,E1 6811.427,E2 6811.427} C_VEL
LIN {X 0,Y 475.016,Z 370.16,A -85,B 0,C 180,E1 6814.22,E2 6814.22} C_VEL
LIN {X 0,Y 484.202,Z 403.318,A -85,B 0,C 180,E1 6815.402,E2 6815.402} C_VEL
LIN {X 0,Y 483.17,Z 437.397,A -85,B 0,C 180,E1 6816.697,E2 6816.697} C_VEL
LIN {X 0,Y 481.662,Z 469.588,A -85,B 0,C 180,E1 6818.688,E2 6818.688} C_VEL
LIN {X 0,Y 479.984,Z 496.565,A -85,B 0,C 180,E1 6821.119,E2 6821.119} C_VEL
LIN {X 0,Y 478.482,Z 521.045,A -85,B 0,C 180,E1 6824.239,E2 6824.239} C_VEL
LIN {X 0,Y 477.21,Z 540.876,A -85,B 0,C 180,E1 6827.866,E2 6827.866} C_VEL
LIN {X 0,Y 476.471,Z 554.983,A -85,B 0,C 180,E1 6831.778,E2 6831.778} C_VEL
LIN {X 0,Y 476.128,Z 562.786,A -85,B 0,C 180,E1 6835.44,E2 6835.44} C_VEL
LIN {X 0,Y 476.063,Z 565.494,A -85,B 0,C 180,E1 6838.176,E2 6838.176} C_VEL
LIN {X 0,Y 475.947,Z 565.308,A -85,B 0,C 180,E1 6841.822,E2 6841.822} C_VEL
LIN {X 0,Y 476.192,Z 560.714,A -85,B 0,C 180,E1 6845.472,E2 6845.472} C_VEL
LIN {X 0,Y 476.543,Z 550.221,A -85,B 0,C 180,E1 6849.468,E2 6849.468} C_VEL
LIN {X 0,Y 477.345,Z 534.07,A -85,B 0,C 180,E1 6853.292,E2 6853.292} C_VEL
LIN {X 0,Y 478.856,Z 512.605,A -85,B 0,C 180,E1 6856.766,E2 6856.766} C_VEL
LIN {X 0,Y 480.561,Z 487.066,A -85,B 0,C 180,E1 6859.711,E2 6859.711} C_VEL
LIN {X 0,Y 482.373,Z 457.4,A -85,B 0,C 180,E1 6862.123,E2 6862.123} C_VEL
LIN {X 0,Y 483.957,Z 425.545,A -85,B 0,C 180,E1 6863.872,E2 6863.872} C_VEL
LIN {X 0,Y 484.146,Z 400.144,A -85,B 0,C 180,E1 6864.802,E2 6864.802} C_VEL
LIN {X 0,Y 474.985,Z 370.16,A -85,B 0,C 180,E1 6865.932,E2 6865.932} C_VEL
LIN {X 0,Y 474.752,Z 370.16,A -85,B 0,C 180,E1 6872.825,E2 6872.825} C_VEL
LIN {X 0,Y 474.796,Z 370.16,A -85,B 0,C 180,E1 6877.287,E2 6877.287} C_VEL
LIN {X 0,Y 474.665,Z 370.16,A -85,B 0,C 180,E1 6882.817,E2 6882.817} C_VEL
LIN {X 0,Y 474.677,Z 370.16,A -85,B 0,C 180,E1 6887.954,E2 6887.954} C_VEL
LIN {X 0,Y 474.7,Z 370.16,A -85,B 0,C 180,E1 6892.871,E2 6892.871} C_VEL
LIN {X 0,Y 474.782,Z 370.16,A -85,B 0,C 180,E1 6899.419,E2 6899.419} C_VEL
LIN {X 0,Y 474.919,Z 370.16,A -85,B 0,C 180,E1 6902.443,E2 6902.443} C_VEL
LIN {X 0,Y 489.161,Z 406.239,A -85,B 0,C 180,E1 6904.211,E2 6904.211} C_VEL
LIN {X 0,Y 487.432,Z 438.784,A -85,B 0,C 180,E1 6905.553,E2 6905.553} C_VEL
LIN {X 0,Y 485.019,Z 468.494,A -85,B 0,C 180,E1 6907.488,E2 6907.488} C_VEL
LIN {X 0,Y 482.368,Z 495.549,A -85,B 0,C 180,E1 6910.037,E2 6910.037} C_VEL
LIN {X 0,Y 479.762,Z 519.926,A -85,B 0,C 180,E1 6913.268,E2 6913.268} C_VEL
LIN {X 0,Y 477.855,Z 539.364,A -85,B 0,C 180,E1 6916.957,E2 6916.957} C_VEL
LIN {X 0,Y 476.698,Z 553.341,A -85,B 0,C 180,E1 6920.866,E2 6920.866} C_VEL
LIN {X 0,Y 476.187,Z 561.466,A -85,B 0,C 180,E1 6924.53,E2 6924.53} C_VEL
LIN {X 0,Y 475.956,Z 565.377,A -85,B 0,C 180,E1 6928.18,E2 6928.18} C_VEL
LIN {X 0,Y 475.964,Z 565.326,A -85,B 0,C 180,E1 6931.825,E2 6931.825} C_VEL
LIN {X 0,Y 476.224,Z 561.311,A -85,B 0,C 180,E1 6935.475,E2 6935.475} C_VEL
LIN {X 0,Y 476.814,Z 551.809,A -85,B 0,C 180,E1 6939.567,E2 6939.567} C_VEL
LIN {X 0,Y 478.056,Z 536.897,A -85,B 0,C 180,E1 6943.509,E2 6943.509} C_VEL
LIN {X 0,Y 480.033,Z 517.778,A -85,B 0,C 180,E1 6946.964,E2 6946.964} C_VEL
LIN {X 0,Y 482.469,Z 494.661,A -85,B 0,C 180,E1 6949.972,E2 6949.972} C_VEL
LIN {X 0,Y 485.153,Z 466.883,A -85,B 0,C 180,E1 6952.544,E2 6952.544} C_VEL
LIN {X 0,Y 487.577,Z 436.207,A -85,B 0,C 180,E1 6954.495,E2 6954.495} C_VEL
LIN {X 0,Y 488.608,Z 404.165,A -85,B 0,C 180,E1 6955.797,E2 6955.797} C_VEL
LIN {X 0,Y 474.863,Z 370.16,A -85,B 0,C 180,E1 6957.556,E2 6957.556} C_VEL
LIN {X 0,Y 474.66,Z 370.16,A -85,B 0,C 180,E1 6963.98,E2 6963.98} C_VEL
LIN {X 0,Y 474.552,Z 370.16,A -85,B 0,C 180,E1 6970.038,E2 6970.038} C_VEL
LIN {X 0,Y 474.635,Z 370.16,A -85,B 0,C 180,E1 6975.437,E2 6975.437} C_VEL
LIN {X 0,Y 474.635,Z 370.16,A -85,B 0,C 180,E1 6980.364,E2 6980.364} C_VEL
LIN {X 0,Y 474.636,Z 370.16,A -85,B 0,C 180,E1 6986.033,E2 6986.033} C_VEL
LIN {X 0,Y 474.779,Z 370.16,A -85,B 0,C 180,E1 6991.427,E2 6991.427} C_VEL
LIN {X 0,Y 475.004,Z 370.16,A -85,B 0,C 180,E1 6997.568,E2 6997.568} C_VEL
LIN {X 0,Y 475.152,Z 370.16,A -85,B 0,C 180,E1 7003.338,E2 7003.338} C_VEL
LIN {X 0,Y 475.268,Z 370.16,A -85,B 0,C 180,E1 7008.983,E2 7008.983} C_VEL
LIN {X 0,Y 475.403,Z 370.16,A -85,B 0,C 180,E1 7014.519,E2 7014.519} C_VEL
LIN {X 0,Y 475.587,Z 370.16,A -85,B 0,C 180,E1 7020.001,E2 7020.001} C_VEL
LIN {X 0,Y 475.437,Z 370.16,A -85,B 0,C 180,E1 7025.483,E2 7025.483} C_VEL
LIN {X 0,Y 475.227,Z 370.16,A -85,B 0,C 180,E1 7031.02,E2 7031.02} C_VEL
LIN {X 0,Y 475.051,Z 370.16,A -85,B 0,C 180,E1 7037.038,E2 7037.038} C_VEL
LIN {X 0,Y 475.001,Z 370.16,A -85,B 0,C 180,E1 7042.487,E2 7042.487} C_VEL
LIN {X 0,Y 474.781,Z 370.16,A -85,B 0,C 180,E1 7048.576,E2 7048.576} C_VEL
LIN {X 0,Y 474.732,Z 370.16,A -85,B 0,C 180,E1 7055.032,E2 7055.032} C_VEL
LIN {X 0,Y 474.664,Z 370.16,A -85,B 0,C 180,E1 7060.047,E2 7060.047} C_VEL
LIN {X 0,Y 474.656,Z 370.16,A -85,B 0,C 180,E1 7065.433,E2 7065.433} C_VEL
LIN {X 0,Y 474.615,Z 370.16,A -85,B 0,C 180,E1 7071.996,E2 7071.996} C_VEL
LIN {X 0,Y 474.711,Z 370.16,A -85,B 0,C 180,E1 7076.064,E2 7076.064} C_VEL
LIN {X 0,Y 474.859,Z 373.198,A -85,B 0,C 180,E1 7076.819,E2 7076.819} C_VEL
LIN {X 0,Y 475.64,Z 383.903,A -85,B 0,C 180,E1 7077.51,E2 7077.51} C_VEL
LIN {X 0,Y 478.639,Z 400.766,A -85,B 0,C 180,E1 7078.029,E2 7078.029} C_VEL
LIN {X 0,Y 483.133,Z 413.885,A -85,B 0,C 180,E1 7078.542,E2 7078.542} C_VEL
LIN {X 0,Y 481.489,Z 452.646,A -85,B 0,C 180,E1 7079.545,E2 7079.545} C_VEL
LIN {X 0,Y 479.214,Z 489.7,A -85,B 0,C 180,E1 7081.232,E2 7081.232} C_VEL
LIN {X 0,Y 476.45,Z 524.325,A -85,B 0,C 180,E1 7083.583,E2 7083.583} C_VEL
LIN {X 0,Y 473.726,Z 556.039,A -85,B 0,C 180,E1 7086.576,E2 7086.576} C_VEL
LIN {X 0,Y 471.402,Z 583.138,A -85,B 0,C 180,E1 7090.045,E2 7090.045} C_VEL
LIN {X 0,Y 469.548,Z 606.21,A -85,B 0,C 180,E1 7094.091,E2 7094.091} C_VEL
LIN {X 0,Y 468.486,Z 623.44,A -85,B 0,C 180,E1 7098.345,E2 7098.345} C_VEL
LIN {X 0,Y 468.068,Z 634.701,A -85,B 0,C 180,E1 7102.564,E2 7102.564} C_VEL
LIN {X 0,Y 467.921,Z 640.159,A -85,B 0,C 180,E1 7106.287,E2 7106.287} C_VEL
LIN {X 0,Y 467.872,Z 642,A -85,B 0,C 180,E1 7109.997,E2 7109.997} C_VEL
LIN {X 0,Y 467.953,Z 639.176,A -85,B 0,C 180,E1 7114.636,E2 7114.636} C_VEL
LIN {X 0,Y 468.225,Z 631.574,A -85,B 0,C 180,E1 7118.832,E2 7118.832} C_VEL
LIN {X 0,Y 468.759,Z 618.424,A -85,B 0,C 180,E1 7123.063,E2 7123.063} C_VEL
LIN {X 0,Y 469.923,Z 600.38,A -85,B 0,C 180,E1 7127.057,E2 7127.057} C_VEL
LIN {X 0,Y 471.914,Z 576.454,A -85,B 0,C 180,E1 7130.91,E2 7130.91} C_VEL
LIN {X 0,Y 474.499,Z 546.98,A -85,B 0,C 180,E1 7134.377,E2 7134.377} C_VEL
LIN {X 0,Y 477.257,Z 515.324,A -85,B 0,C 180,E1 7137.104,E2 7137.104} C_VEL
LIN {X 0,Y 479.934,Z 479.387,A -85,B 0,C 180,E1 7139.318,E2 7139.318} C_VEL
LIN {X 0,Y 482.052,Z 441.695,A -85,B 0,C 180,E1 7140.812,E2 7140.812} C_VEL
LIN {X 0,Y 482.612,Z 409.901,A -85,B 0,C 180,E1 7141.562,E2 7141.562} C_VEL
LIN {X 0,Y 466.985,Z 370.16,A -85,B 0,C 180,E1 7143.37,E2 7143.37} C_VEL
LIN {X 0,Y 466.659,Z 370.16,A -85,B 0,C 180,E1 7150.45,E2 7150.45} C_VEL
LIN {X 0,Y 466.574,Z 370.16,A -85,B 0,C 180,E1 7157.046,E2 7157.046} C_VEL
LIN {X 0,Y 466.625,Z 370.16,A -85,B 0,C 180,E1 7161.943,E2 7161.943} C_VEL
LIN {X 0,Y 466.789,Z 370.16,A -85,B 0,C 180,E1 7168.739,E2 7168.739} C_VEL
LIN {X 0,Y 467.071,Z 370.924,A -85,B 0,C 180,E1 7173.794,E2 7173.794} C_VEL
LIN {X 0,Y 476.908,Z 403.884,A -85,B 0,C 180,E1 7175.049,E2 7175.049} C_VEL
LIN {X 0,Y 475.797,Z 438.337,A -85,B 0,C 180,E1 7176.376,E2 7176.376} C_VEL
LIN {X 0,Y 474.193,Z 470.565,A -85,B 0,C 180,E1 7178.41,E2 7178.41} C_VEL
LIN {X 0,Y 472.276,Z 499.087,A -85,B 0,C 180,E1 7181.051,E2 7181.051} C_VEL
LIN {X 0,Y 470.781,Z 522.548,A -85,B 0,C 180,E1 7184.137,E2 7184.137} C_VEL
LIN {X 0,Y 469.439,Z 541.45,A -85,B 0,C 180,E1 7187.662,E2 7187.662} C_VEL
LIN {X 0,Y 468.659,Z 555.61,A -85,B 0,C 180,E1 7191.64,E2 7191.64} C_VEL
LIN {X 0,Y 468.293,Z 563.45,A -85,B 0,C 180,E1 7195.363,E2 7195.363} C_VEL
LIN {X 0,Y 468.205,Z 566.16,A -85,B 0,C 180,E1 7198.146,E2 7198.146} C_VEL
LIN {X 0,Y 468.083,Z 565.944,A -85,B 0,C 180,E1 7201.852,E2 7201.852} C_VEL
LIN {X 0,Y 468.325,Z 561.294,A -85,B 0,C 180,E1 7205.564,E2 7205.564} C_VEL
LIN {X 0,Y 468.717,Z 551.781,A -85,B 0,C 180,E1 7209.292,E2 7209.292} C_VEL
LIN {X 0,Y 469.46,Z 536.798,A -85,B 0,C 180,E1 7213.045,E2 7213.045} C_VEL
LIN {X 0,Y 470.986,Z 516.274,A -85,B 0,C 180,E1 7216.55,E2 7216.55} C_VEL
LIN {X 0,Y 472.665,Z 491.814,A -85,B 0,C 180,E1 7219.547,E2 7219.547} C_VEL
LIN {X 0,Y 474.572,Z 462.791,A -85,B 0,C 180,E1 7222.085,E2 7222.085} C_VEL
LIN {X 0,Y 476.396,Z 430.012,A -85,B 0,C 180,E1 7224.025,E2 7224.025} C_VEL
LIN {X 0,Y 476.673,Z 401.416,A -85,B 0,C 180,E1 7225.127,E2 7225.127} C_VEL
LIN {X 0,Y 467.046,Z 370.16,A -85,B 0,C 180,E1 7226.32,E2 7226.32} C_VEL
LIN {X 0,Y 466.82,Z 370.16,A -85,B 0,C 180,E1 7233.456,E2 7233.456} C_VEL
LIN {X 0,Y 466.763,Z 370.16,A -85,B 0,C 180,E1 7240.441,E2 7240.441} C_VEL
LIN {X 0,Y 466.785,Z 370.16,A -85,B 0,C 180,E1 7247.075,E2 7247.075} C_VEL
LIN {X 0,Y 466.719,Z 370.16,A -85,B 0,C 180,E1 7251.956,E2 7251.956} C_VEL
LIN {X 0,Y 466.785,Z 370.16,A -85,B 0,C 180,E1 7258.743,E2 7258.743} C_VEL
LIN {X 0,Y 466.975,Z 370.711,A -85,B 0,C 180,E1 7261.892,E2 7261.892} C_VEL
LIN {X 0,Y 482.038,Z 407.266,A -85,B 0,C 180,E1 7263.771,E2 7263.771} C_VEL
LIN {X 0,Y 480.345,Z 440.03,A -85,B 0,C 180,E1 7265.169,E2 7265.169} C_VEL
LIN {X 0,Y 477.727,Z 470.822,A -85,B 0,C 180,E1 7267.232,E2 7267.232} C_VEL
LIN {X 0,Y 474.767,Z 498.578,A -85,B 0,C 180,E1 7269.961,E2 7269.961} C_VEL
LIN {X 0,Y 472.043,Z 522.135,A -85,B 0,C 180,E1 7273.226,E2 7273.226} C_VEL
LIN {X 0,Y 470.093,Z 541.147,A -85,B 0,C 180,E1 7276.974,E2 7276.974} C_VEL
LIN {X 0,Y 468.855,Z 555.294,A -85,B 0,C 180,E1 7281.18,E2 7281.18} C_VEL
LIN {X 0,Y 468.29,Z 563.5,A -85,B 0,C 180,E1 7285.367,E2 7285.367} C_VEL
LIN {X 0,Y 468.145,Z 566.516,A -85,B 0,C 180,E1 7290.003,E2 7290.003} C_VEL
LIN {X 0,Y 468.304,Z 563.382,A -85,B 0,C 180,E1 7294.638,E2 7294.638} C_VEL
LIN {X 0,Y 468.875,Z 555.04,A -85,B 0,C 180,E1 7298.825,E2 7298.825} C_VEL
LIN {X 0,Y 470.124,Z 540.728,A -85,B 0,C 180,E1 7303.03,E2 7303.03} C_VEL
LIN {X 0,Y 472.162,Z 521.568,A -85,B 0,C 180,E1 7306.775,E2 7306.775} C_VEL
LIN {X 0,Y 474.889,Z 497.447,A -85,B 0,C 180,E1 7310.077,E2 7310.077} C_VEL
LIN {X 0,Y 477.82,Z 469.26,A -85,B 0,C 180,E1 7312.801,E2 7312.801} C_VEL
LIN {X 0,Y 480.372,Z 438.969,A -85,B 0,C 180,E1 7314.8,E2 7314.8} C_VEL
LIN {X 0,Y 481.719,Z 406.659,A -85,B 0,C 180,E1 7316.177,E2 7316.177} C_VEL
LIN {X 0,Y 466.895,Z 370.16,A -85,B 0,C 180,E1 7318.113,E2 7318.113} C_VEL
LIN {X 0,Y 466.752,Z 370.16,A -85,B 0,C 180,E1 7323.467,E2 7323.467} C_VEL
LIN {X 0,Y 466.62,Z 370.16,A -85,B 0,C 180,E1 7330.462,E2 7330.462} C_VEL
LIN {X 0,Y 466.759,Z 370.16,A -85,B 0,C 180,E1 7337.07,E2 7337.07} C_VEL
LIN {X 0,Y 466.68,Z 370.16,A -85,B 0,C 180,E1 7341.951,E2 7341.951} C_VEL
LIN {X 0,Y 466.733,Z 370.16,A -85,B 0,C 180,E1 7348.738,E2 7348.738} C_VEL
LIN {X 0,Y 467.036,Z 370.16,A -85,B 0,C 180,E1 7355.188,E2 7355.188} C_VEL
LIN {X 0,Y 467.149,Z 370.16,A -85,B 0,C 180,E1 7361.092,E2 7361.092} C_VEL
LIN {X 0,Y 467.308,Z 370.16,A -85,B 0,C 180,E1 7366.894,E2 7366.894} C_VEL
LIN {X 0,Y 467.404,Z 370.16,A -85,B 0,C 180,E1 7372.557,E2 7372.557} C_VEL
LIN {X 0,Y 467.569,Z 370.16,A -85,B 0,C 180,E1 7378.146,E2 7378.146} C_VEL
LIN {X 0,Y 467.51,Z 370.16,A -85,B 0,C 180,E1 7383.715,E2 7383.715} C_VEL
LIN {X 0,Y 467.356,Z 370.16,A -85,B 0,C 180,E1 7389.322,E2 7389.322} C_VEL
LIN {X 0,Y 467.201,Z 370.16,A -85,B 0,C 180,E1 7395.026,E2 7395.026} C_VEL
LIN {X 0,Y 467.086,Z 370.16,A -85,B 0,C 180,E1 7400.888,E2 7400.888} C_VEL
LIN {X 0,Y 466.923,Z 370.16,A -85,B 0,C 180,E1 7406.997,E2 7406.997} C_VEL
LIN {X 0,Y 466.785,Z 370.16,A -85,B 0,C 180,E1 7413.461,E2 7413.461} C_VEL
LIN {X 0,Y 466.724,Z 370.16,A -85,B 0,C 180,E1 7420.448,E2 7420.448} C_VEL
LIN {X 0,Y 466.774,Z 370.16,A -85,B 0,C 180,E1 7427.066,E2 7427.066} C_VEL
LIN {X 0,Y 466.711,Z 370.16,A -85,B 0,C 180,E1 7431.948,E2 7431.948} C_VEL
LIN {X 0,Y 466.848,Z 370.16,A -85,B 0,C 180,E1 7436.663,E2 7436.663} C_VEL
LIN {X 0,Y 478.639,Z 400.766,A -85,B 0,C 180,E1 7438.029,E2 7438.029} C_VEL
LIN {X 0,Y 479.61,Z 411.42,A -85,B 0,C 180,E1 7438.279,E2 7438.279} C_VEL
LIN {X 0,Y 475.301,Z 435.777,A -85,B 0,C 180,E1 7438.6,E2 7438.6} C_VEL
LIN {X 0,Y 473.067,Z 473.137,A -85,B 0,C 180,E1 7440.01,E2 7440.01} C_VEL
LIN {X 0,Y 470.203,Z 510.172,A -85,B 0,C 180,E1 7442.188,E2 7442.188} C_VEL
LIN {X 0,Y 467.257,Z 543.021,A -85,B 0,C 180,E1 7444.958,E2 7444.958} C_VEL
LIN {X 0,Y 464.559,Z 571.799,A -85,B 0,C 180,E1 7448.258,E2 7448.258} C_VEL
LIN {X 0,Y 462.51,Z 595.655,A -85,B 0,C 180,E1 7451.934,E2 7451.934} C_VEL
LIN {X 0,Y 461.116,Z 615.166,A -85,B 0,C 180,E1 7456.062,E2 7456.062} C_VEL
LIN {X 0,Y 460.359,Z 629.649,A -85,B 0,C 180,E1 7460.533,E2 7460.533} C_VEL
LIN {X 0,Y 460.076,Z 637.375,A -85,B 0,C 180,E1 7464.332,E2 7464.332} C_VEL
LIN {X 0,Y 459.997,Z 641.097,A -85,B 0,C 180,E1 7468.111,E2 7468.111} C_VEL
LIN {X 0,Y 460.032,Z 641.102,A -85,B 0,C 180,E1 7471.883,E2 7471.883} C_VEL
LIN {X 0,Y 460.036,Z 637.381,A -85,B 0,C 180,E1 7475.663,E2 7475.663} C_VEL
LIN {X 0,Y 460.387,Z 628.444,A -85,B 0,C 180,E1 7479.939,E2 7479.939} C_VEL
LIN {X 0,Y 461.156,Z 613.818,A -85,B 0,C 180,E1 7484.272,E2 7484.272} C_VEL
LIN {X 0,Y 462.654,Z 593.823,A -85,B 0,C 180,E1 7488.384,E2 7488.384} C_VEL
LIN {X 0,Y 464.712,Z 569.747,A -85,B 0,C 180,E1 7492.011,E2 7492.011} C_VEL
LIN {X 0,Y 467.597,Z 539.381,A -85,B 0,C 180,E1 7495.401,E2 7495.401} C_VEL
LIN {X 0,Y 470.601,Z 505.571,A -85,B 0,C 180,E1 7498.124,E2 7498.124} C_VEL
LIN {X 0,Y 473.375,Z 469.367,A -85,B 0,C 180,E1 7500.169,E2 7500.169} C_VEL
LIN {X 0,Y 475.575,Z 431.279,A -85,B 0,C 180,E1 7501.513,E2 7501.513} C_VEL
LIN {X 0,Y 475.515,Z 411.969,A -85,B 0,C 180,E1 7501.972,E2 7501.972} C_VEL
LIN {X 0,Y 458.974,Z 370.16,A -85,B 0,C 180,E1 7503.971,E2 7503.971} C_VEL
LIN {X 0,Y 458.757,Z 370.16,A -85,B 0,C 180,E1 7510.622,E2 7510.622} C_VEL
LIN {X 0,Y 458.647,Z 370.16,A -85,B 0,C 180,E1 7516.564,E2 7516.564} C_VEL
LIN {X 0,Y 458.705,Z 370.16,A -85,B 0,C 180,E1 7522.378,E2 7522.378} C_VEL
LIN {X 0,Y 458.871,Z 370.16,A -85,B 0,C 180,E1 7529.066,E2 7529.066} C_VEL
LIN {X 0,Y 459.098,Z 370.342,A -85,B 0,C 180,E1 7533.29,E2 7533.29} C_VEL
LIN {X 0,Y 469.534,Z 404.633,A -85,B 0,C 180,E1 7534.672,E2 7534.672} C_VEL
LIN {X 0,Y 468.475,Z 439.364,A -85,B 0,C 180,E1 7536.047,E2 7536.047} C_VEL
LIN {X 0,Y 466.795,Z 470.802,A -85,B 0,C 180,E1 7538.051,E2 7538.051} C_VEL
LIN {X 0,Y 464.857,Z 498.59,A -85,B 0,C 180,E1 7540.635,E2 7540.635} C_VEL
LIN {X 0,Y 463.131,Z 523.065,A -85,B 0,C 180,E1 7543.867,E2 7543.867} C_VEL
LIN {X 0,Y 461.677,Z 542.048,A -85,B 0,C 180,E1 7547.452,E2 7547.452} C_VEL
LIN {X 0,Y 460.845,Z 556.276,A -85,B 0,C 180,E1 7551.498,E2 7551.498} C_VEL
LIN {X 0,Y 460.442,Z 564.117,A -85,B 0,C 180,E1 7555.284,E2 7555.284} C_VEL
LIN {X 0,Y 460.355,Z 566.829,A -85,B 0,C 180,E1 7558.114,E2 7558.114} C_VEL
LIN {X 0,Y 460.21,Z 566.581,A -85,B 0,C 180,E1 7561.884,E2 7561.884} C_VEL
LIN {X 0,Y 460.477,Z 561.869,A -85,B 0,C 180,E1 7565.659,E2 7565.659} C_VEL
LIN {X 0,Y 460.893,Z 551.108,A -85,B 0,C 180,E1 7569.809,E2 7569.809} C_VEL
LIN {X 0,Y 461.865,Z 534.865,A -85,B 0,C 180,E1 7573.719,E2 7573.719} C_VEL
LIN {X 0,Y 463.549,Z 512.894,A -85,B 0,C 180,E1 7577.337,E2 7577.337} C_VEL
LIN {X 0,Y 465.518,Z 486.449,A -85,B 0,C 180,E1 7580.412,E2 7580.412} C_VEL
LIN {X 0,Y 467.602,Z 456.497,A -85,B 0,C 180,E1 7582.861,E2 7582.861} C_VEL
LIN {X 0,Y 469.31,Z 423.384,A -85,B 0,C 180,E1 7584.665,E2 7584.665} C_VEL
LIN {X 0,Y 469.339,Z 403.309,A -85,B 0,C 180,E1 7585.427,E2 7585.427} C_VEL
LIN {X 0,Y 459.081,Z 370.16,A -85,B 0,C 180,E1 7586.753,E2 7586.753} C_VEL
LIN {X 0,Y 458.909,Z 370.16,A -85,B 0,C 180,E1 7591.857,E2 7591.857} C_VEL
LIN {X 0,Y 458.887,Z 370.16,A -85,B 0,C 180,E1 7598.815,E2 7598.815} C_VEL
LIN {X 0,Y 458.856,Z 370.16,A -85,B 0,C 180,E1 7603.855,E2 7603.855} C_VEL
LIN {X 0,Y 458.843,Z 370.16,A -85,B 0,C 180,E1 7609.362,E2 7609.362} C_VEL
LIN {X 0,Y 458.787,Z 370.16,A -85,B 0,C 180,E1 7615.88,E2 7615.88} C_VEL
LIN {X 0,Y 459.023,Z 370.734,A -85,B 0,C 180,E1 7621.297,E2 7621.297} C_VEL
LIN {X 0,Y 474.539,Z 408.103,A -85,B 0,C 180,E1 7623.285,E2 7623.285} C_VEL
LIN {X 0,Y 473.535,Z 438.237,A -85,B 0,C 180,E1 7624.607,E2 7624.607} C_VEL
LIN {X 0,Y 470.722,Z 469.291,A -85,B 0,C 180,E1 7626.66,E2 7626.66} C_VEL
LIN {X 0,Y 467.692,Z 496.663,A -85,B 0,C 180,E1 7629.304,E2 7629.304} C_VEL
LIN {X 0,Y 464.85,Z 520.031,A -85,B 0,C 180,E1 7632.47,E2 7632.47} C_VEL
LIN {X 0,Y 462.501,Z 539.843,A -85,B 0,C 180,E1 7636.275,E2 7636.275} C_VEL
LIN {X 0,Y 461.261,Z 552.986,A -85,B 0,C 180,E1 7639.935,E2 7639.935} C_VEL
LIN {X 0,Y 460.508,Z 562.791,A -85,B 0,C 180,E1 7644.343,E2 7644.343} C_VEL
LIN {X 0,Y 460.219,Z 566.657,A -85,B 0,C 180,E1 7648.118,E2 7648.118} C_VEL
LIN {X 0,Y 460.228,Z 566.607,A -85,B 0,C 180,E1 7651.888,E2 7651.888} C_VEL
LIN {X 0,Y 460.545,Z 562.64,A -85,B 0,C 180,E1 7655.662,E2 7655.662} C_VEL
LIN {X 0,Y 461.278,Z 552.678,A -85,B 0,C 180,E1 7660.077,E2 7660.077} C_VEL
LIN {X 0,Y 462.778,Z 537.364,A -85,B 0,C 180,E1 7664.206,E2 7664.206} C_VEL
LIN {X 0,Y 465.301,Z 516.368,A -85,B 0,C 180,E1 7668.008,E2 7668.008} C_VEL
LIN {X 0,Y 468.329,Z 491.215,A -85,B 0,C 180,E1 7671.204,E2 7671.204} C_VEL
LIN {X 0,Y 471.414,Z 462.838,A -85,B 0,C 180,E1 7673.748,E2 7673.748} C_VEL
LIN {X 0,Y 474.014,Z 430.729,A -85,B 0,C 180,E1 7675.676,E2 7675.676} C_VEL
LIN {X 0,Y 474.535,Z 408.221,A -85,B 0,C 180,E1 7676.618,E2 7676.618} C_VEL
LIN {X 0,Y 459.874,Z 373.818,A -85,B 0,C 180,E1 7678.493,E2 7678.493} C_VEL
LIN {X 0,Y 458.959,Z 370.16,A -85,B 0,C 180,E1 7678.689,E2 7678.689} C_VEL
LIN {X 0,Y 458.754,Z 370.16,A -85,B 0,C 180,E1 7684.413,E2 7684.413} C_VEL
LIN {X 0,Y 458.695,Z 370.16,A -85,B 0,C 180,E1 7691.311,E2 7691.311} C_VEL
LIN {X 0,Y 458.821,Z 370.16,A -85,B 0,C 180,E1 7696.549,E2 7696.549} C_VEL
LIN {X 0,Y 458.748,Z 370.16,A -85,B 0,C 180,E1 7702.38,E2 7702.38} C_VEL
LIN {X 0,Y 458.82,Z 370.16,A -85,B 0,C 180,E1 7709.087,E2 7709.087} C_VEL
LIN {X 0,Y 459.043,Z 370.16,A -85,B 0,C 180,E1 7714.614,E2 7714.614} C_VEL
LIN {X 0,Y 459.241,Z 370.16,A -85,B 0,C 180,E1 7720.754,E2 7720.754} C_VEL
LIN {X 0,Y 459.411,Z 370.16,A -85,B 0,C 180,E1 7726.665,E2 7726.665} C_VEL
LIN {X 0,Y 459.491,Z 370.16,A -85,B 0,C 180,E1 7732.428,E2 7732.428} C_VEL
LIN {X 0,Y 459.668,Z 370.16,A -85,B 0,C 180,E1 7738.114,E2 7738.114} C_VEL
LIN {X 0,Y 459.602,Z 370.16,A -85,B 0,C 180,E1 7743.779,E2 7743.779} C_VEL
LIN {X 0,Y 459.445,Z 370.16,A -85,B 0,C 180,E1 7749.484,E2 7749.484} C_VEL
LIN {X 0,Y 459.266,Z 370.16,A -85,B 0,C 180,E1 7755.292,E2 7755.292} C_VEL
LIN {X 0,Y 459.135,Z 370.16,A -85,B 0,C 180,E1 7761.268,E2 7761.268} C_VEL
LIN {X 0,Y 458.972,Z 370.16,A -85,B 0,C 180,E1 7767.504,E2 7767.504} C_VEL
LIN {X 0,Y 458.81,Z 370.16,A -85,B 0,C 180,E1 7774.414,E2 7774.414} C_VEL
LIN {X 0,Y 458.842,Z 370.16,A -85,B 0,C 180,E1 7780.631,E2 7780.631} C_VEL
LIN {X 0,Y 458.837,Z 370.16,A -85,B 0,C 180,E1 7786.544,E2 7786.544} C_VEL
LIN {X 0,Y 458.78,Z 370.16,A -85,B 0,C 180,E1 7792.372,E2 7792.372} C_VEL
LIN {X 0,Y 458.852,Z 370.16,A -85,B 0,C 180,E1 7796.079,E2 7796.079} C_VEL
LIN {X 0,Y 476.077,Z 415.05,A -85,B 0,C 180,E1 7798.129,E2 7798.129} C_VEL
LIN {X 0,Y 475.301,Z 435.777,A -85,B 0,C 180,E1 7798.6,E2 7798.6} C_VEL
LIN {X 0,Y 466.441,Z 466.926,A -85,B 0,C 180,E1 7799.302,E2 7799.302} C_VEL
LIN {X 0,Y 466.21,Z 468.962,A -85,B 0,C 180,E1 7799.395,E2 7799.395} C_VEL
LIN {X 0,Y 463.22,Z 505.189,A -85,B 0,C 180,E1 7801.491,E2 7801.491} C_VEL
LIN {X 0,Y 460.132,Z 539.085,A -85,B 0,C 180,E1 7804.282,E2 7804.282} C_VEL
LIN {X 0,Y 457.115,Z 568.894,A -85,B 0,C 180,E1 7807.656,E2 7807.656} C_VEL
LIN {X 0,Y 454.796,Z 593.655,A -85,B 0,C 180,E1 7811.444,E2 7811.444} C_VEL
LIN {X 0,Y 453.275,Z 613.521,A -85,B 0,C 180,E1 7815.604,E2 7815.604} C_VEL
LIN {X 0,Y 452.503,Z 627.707,A -85,B 0,C 180,E1 7819.881,E2 7819.881} C_VEL
LIN {X 0,Y 452.197,Z 636.709,A -85,B 0,C 180,E1 7824.233,E2 7824.233} C_VEL
LIN {X 0,Y 452.126,Z 640.456,A -85,B 0,C 180,E1 7828.078,E2 7828.078} C_VEL
LIN {X 0,Y 452.156,Z 640.461,A -85,B 0,C 180,E1 7831.916,E2 7831.916} C_VEL
LIN {X 0,Y 452.153,Z 636.714,A -85,B 0,C 180,E1 7835.762,E2 7835.762} C_VEL
LIN {X 0,Y 452.504,Z 627.717,A -85,B 0,C 180,E1 7840.113,E2 7840.113} C_VEL
LIN {X 0,Y 453.294,Z 613.481,A -85,B 0,C 180,E1 7844.405,E2 7844.405} C_VEL
LIN {X 0,Y 454.891,Z 592.765,A -85,B 0,C 180,E1 7848.709,E2 7848.709} C_VEL
LIN {X 0,Y 457.268,Z 567.412,A -85,B 0,C 180,E1 7852.539,E2 7852.539} C_VEL
LIN {X 0,Y 460.247,Z 536.458,A -85,B 0,C 180,E1 7855.967,E2 7855.967} C_VEL
LIN {X 0,Y 463.484,Z 502.35,A -85,B 0,C 180,E1 7858.705,E2 7858.705} C_VEL
LIN {X 0,Y 466.5,Z 465.6,A -85,B 0,C 180,E1 7860.755,E2 7860.755} C_VEL
LIN {X 0,Y 468.689,Z 429.076,A -85,B 0,C 180,E1 7862.016,E2 7862.016} C_VEL
LIN {X 0,Y 468.425,Z 414.003,A -85,B 0,C 180,E1 7862.398,E2 7862.398} C_VEL
LIN {X 0,Y 451.02,Z 370.16,A -85,B 0,C 180,E1 7864.564,E2 7864.564} C_VEL
LIN {X 0,Y 450.844,Z 370.16,A -85,B 0,C 180,E1 7869.64,E2 7869.64} C_VEL
LIN {X 0,Y 450.67,Z 370.16,A -85,B 0,C 180,E1 7875.133,E2 7875.133} C_VEL
LIN {X 0,Y 450.762,Z 370.16,A -85,B 0,C 180,E1 7880.572,E2 7880.572} C_VEL
LIN {X 0,Y 450.842,Z 370.16,A -85,B 0,C 180,E1 7887.082,E2 7887.082} C_VEL
LIN {X 0,Y 451.119,Z 370.16,A -85,B 0,C 180,E1 7892.744,E2 7892.744} C_VEL
LIN {X 0,Y 462.195,Z 405.504,A -85,B 0,C 180,E1 7894.277,E2 7894.277} C_VEL
LIN {X 0,Y 461.125,Z 441.324,A -85,B 0,C 180,E1 7895.743,E2 7895.743} C_VEL
LIN {X 0,Y 459.344,Z 472.728,A -85,B 0,C 180,E1 7897.814,E2 7897.814} C_VEL
LIN {X 0,Y 457.183,Z 501.179,A -85,B 0,C 180,E1 7900.548,E2 7900.548} C_VEL
LIN {X 0,Y 455.414,Z 525.094,A -85,B 0,C 180,E1 7903.834,E2 7903.834} C_VEL
LIN {X 0,Y 453.893,Z 543.751,A -85,B 0,C 180,E1 7907.478,E2 7907.478} C_VEL
LIN {X 0,Y 453.033,Z 556.95,A -85,B 0,C 180,E1 7911.35,E2 7911.35} C_VEL
LIN {X 0,Y 452.603,Z 564.811,A -85,B 0,C 180,E1 7915.202,E2 7915.202} C_VEL
LIN {X 0,Y 452.505,Z 567.506,A -85,B 0,C 180,E1 7918.081,E2 7918.081} C_VEL
LIN {X 0,Y 452.351,Z 567.221,A -85,B 0,C 180,E1 7921.917,E2 7921.917} C_VEL
LIN {X 0,Y 452.632,Z 562.437,A -85,B 0,C 180,E1 7925.757,E2 7925.757} C_VEL
LIN {X 0,Y 453.098,Z 551.568,A -85,B 0,C 180,E1 7929.979,E2 7929.979} C_VEL
LIN {X 0,Y 454.105,Z 535.509,A -85,B 0,C 180,E1 7933.884,E2 7933.884} C_VEL
LIN {X 0,Y 455.802,Z 514.691,A -85,B 0,C 180,E1 7937.392,E2 7937.392} C_VEL
LIN {X 0,Y 457.775,Z 489.397,A -85,B 0,C 180,E1 7940.444,E2 7940.444} C_VEL
LIN {X 0,Y 459.869,Z 459.93,A -85,B 0,C 180,E1 7942.964,E2 7942.964} C_VEL
LIN {X 0,Y 461.761,Z 427.549,A -85,B 0,C 180,E1 7944.837,E2 7944.837} C_VEL
LIN {X 0,Y 461.874,Z 404.521,A -85,B 0,C 180,E1 7945.761,E2 7945.761} C_VEL
LIN {X 0,Y 451.145,Z 370.16,A -85,B 0,C 180,E1 7947.18,E2 7947.18} C_VEL
LIN {X 0,Y 450.899,Z 370.16,A -85,B 0,C 180,E1 7952.929,E2 7952.929} C_VEL
LIN {X 0,Y 450.929,Z 370.16,A -85,B 0,C 180,E1 7959.453,E2 7959.453} C_VEL
LIN {X 0,Y 450.87,Z 370.16,A -85,B 0,C 180,E1 7965.163,E2 7965.163} C_VEL
LIN {X 0,Y 450.882,Z 370.16,A -85,B 0,C 180,E1 7970.555,E2 7970.555} C_VEL
LIN {X 0,Y 450.851,Z 370.16,A -85,B 0,C 180,E1 7977.082,E2 7977.082} C_VEL
LIN {X 0,Y 451.024,Z 370.16,A -85,B 0,C 180,E1 7980.647,E2 7980.647} C_VEL
LIN {X 0,Y 467.179,Z 409.327,A -85,B 0,C 180,E1 7982.806,E2 7982.806} C_VEL
LIN {X 0,Y 468.102,Z 415.885,A -85,B 0,C 180,E1 7983.13,E2 7983.13} C_VEL
LIN {X 0,Y 465.731,Z 448.481,A -85,B 0,C 180,E1 7984.721,E2 7984.721} C_VEL
LIN {X 0,Y 462.616,Z 478.705,A -85,B 0,C 180,E1 7987.008,E2 7987.008} C_VEL
LIN {X 0,Y 459.347,Z 505.22,A -85,B 0,C 180,E1 7989.909,E2 7989.909} C_VEL
LIN {X 0,Y 456.41,Z 528.188,A -85,B 0,C 180,E1 7993.453,E2 7993.453} C_VEL
LIN {X 0,Y 454.265,Z 546.291,A -85,B 0,C 180,E1 7997.492,E2 7997.492} C_VEL
LIN {X 0,Y 453.062,Z 558.934,A -85,B 0,C 180,E1 8001.838,E2 8001.838} C_VEL
LIN {X 0,Y 452.505,Z 565.913,A -85,B 0,C 180,E1 8006.166,E2 8006.166} C_VEL
LIN {X 0,Y 452.4,Z 567.79,A -85,B 0,C 180,E1 8010.003,E2 8010.003} C_VEL
LIN {X 0,Y 452.618,Z 564.681,A -85,B 0,C 180,E1 8014.8,E2 8014.8} C_VEL
LIN {X 0,Y 453.269,Z 556.409,A -85,B 0,C 180,E1 8019.131,E2 8019.131} C_VEL
LIN {X 0,Y 454.731,Z 542.193,A -85,B 0,C 180,E1 8023.48,E2 8023.48} C_VEL
LIN {X 0,Y 457.061,Z 523.12,A -85,B 0,C 180,E1 8027.347,E2 8027.347} C_VEL
LIN {X 0,Y 460.09,Z 499.357,A -85,B 0,C 180,E1 8030.729,E2 8030.729} C_VEL
LIN {X 0,Y 463.266,Z 472.829,A -85,B 0,C 180,E1 8033.418,E2 8033.418} C_VEL
LIN {X 0,Y 466.263,Z 441.509,A -85,B 0,C 180,E1 8035.596,E2 8035.596} C_VEL
LIN {X 0,Y 467.624,Z 410.665,A -85,B 0,C 180,E1 8037.017,E2 8037.017} C_VEL
LIN {X 0,Y 452.944,Z 375.394,A -85,B 0,C 180,E1 8039.002,E2 8039.002} C_VEL
LIN {X 0,Y 450.998,Z 370.16,A -85,B 0,C 180,E1 8039.283,E2 8039.283} C_VEL
LIN {X 0,Y 450.807,Z 370.16,A -85,B 0,C 180,E1 8046.298,E2 8046.298} C_VEL
LIN {X 0,Y 450.758,Z 370.16,A -85,B 0,C 180,E1 8052.365,E2 8052.365} C_VEL
LIN {X 0,Y 450.845,Z 370.16,A -85,B 0,C 180,E1 8057.812,E2 8057.812} C_VEL
LIN {X 0,Y 450.826,Z 370.16,A -85,B 0,C 180,E1 8063.707,E2 8063.707} C_VEL
LIN {X 0,Y 450.903,Z 370.16,A -85,B 0,C 180,E1 8069.761,E2 8069.761} C_VEL
LIN {X 0,Y 451.144,Z 370.16,A -85,B 0,C 180,E1 8076.255,E2 8076.255} C_VEL
LIN {X 0,Y 451.349,Z 370.16,A -85,B 0,C 180,E1 8082.431,E2 8082.431} C_VEL
LIN {X 0,Y 451.49,Z 370.16,A -85,B 0,C 180,E1 8088.395,E2 8088.395} C_VEL
LIN {X 0,Y 451.653,Z 370.16,A -85,B 0,C 180,E1 8094.23,E2 8094.23} C_VEL
LIN {X 0,Y 451.923,Z 370.16,A -85,B 0,C 180,E1 8100.001,E2 8100.001} C_VEL
LIN {X 0,Y 451.721,Z 370.16,A -85,B 0,C 180,E1 8105.772,E2 8105.772} C_VEL
LIN {X 0,Y 451.439,Z 370.16,A -85,B 0,C 180,E1 8111.609,E2 8111.609} C_VEL
LIN {X 0,Y 451.31,Z 370.16,A -85,B 0,C 180,E1 8117.573,E2 8117.573} C_VEL
LIN {X 0,Y 451.142,Z 370.16,A -85,B 0,C 180,E1 8123.748,E2 8123.748} C_VEL
LIN {X 0,Y 450.924,Z 370.16,A -85,B 0,C 180,E1 8130.24,E2 8130.24} C_VEL
LIN {X 0,Y 450.911,Z 370.16,A -85,B 0,C 180,E1 8137.183,E2 8137.183} C_VEL
LIN {X 0,Y 450.848,Z 370.16,A -85,B 0,C 180,E1 8142.371,E2 8142.371} C_VEL
LIN {X 0,Y 450.862,Z 370.16,A -85,B 0,C 180,E1 8147.808,E2 8147.808} C_VEL
LIN {X 0,Y 450.865,Z 370.16,A -85,B 0,C 180,E1 8153.696,E2 8153.696} C_VEL
LIN {X 0,Y 450.919,Z 370.16,A -85,B 0,C 180,E1 8155.469,E2 8155.469} C_VEL
LIN {X 0,Y 469.069,Z 417.249,A -85,B 0,C 180,E1 8157.716,E2 8157.716} C_VEL
LIN {X 0,Y 467.086,Z 455.653,A -85,B 0,C 180,E1 8158.821,E2 8158.821} C_VEL
LIN {X 0,Y 466.21,Z 468.962,A -85,B 0,C 180,E1 8159.395,E2 8159.395} C_VEL
LIN {X 0,Y 461.29,Z 485.086,A -85,B 0,C 180,E1 8160.014,E2 8160.014} C_VEL
LIN {X 0,Y 456.636,Z 498.766,A -85,B 0,C 180,E1 8160.655,E2 8160.655} C_VEL
LIN {X 0,Y 456.41,Z 500.677,A -85,B 0,C 180,E1 8160.784,E2 8160.784} C_VEL
LIN {X 0,Y 453.122,Z 533.69,A -85,B 0,C 180,E1 8163.454,E2 8163.454} C_VEL
LIN {X 0,Y 449.773,Z 565.428,A -85,B 0,C 180,E1 8166.962,E2 8166.962} C_VEL
LIN {X 0,Y 447.225,Z 590.69,A -85,B 0,C 180,E1 8170.771,E2 8170.771} C_VEL
LIN {X 0,Y 445.526,Z 611.488,A -85,B 0,C 180,E1 8175.067,E2 8175.067} C_VEL
LIN {X 0,Y 444.645,Z 626.976,A -85,B 0,C 180,E1 8179.7,E2 8179.7} C_VEL
LIN {X 0,Y 444.318,Z 636.043,A -85,B 0,C 180,E1 8184.13,E2 8184.13} C_VEL
LIN {X 0,Y 444.245,Z 639.815,A -85,B 0,C 180,E1 8188.044,E2 8188.044} C_VEL
LIN {X 0,Y 444.274,Z 639.819,A -85,B 0,C 180,E1 8191.95,E2 8191.95} C_VEL
LIN {X 0,Y 444.273,Z 636.048,A -85,B 0,C 180,E1 8195.865,E2 8195.865} C_VEL
LIN {X 0,Y 444.65,Z 626.986,A -85,B 0,C 180,E1 8200.294,E2 8200.294} C_VEL
LIN {X 0,Y 445.564,Z 611.451,A -85,B 0,C 180,E1 8204.937,E2 8204.937} C_VEL
LIN {X 0,Y 447.277,Z 590.691,A -85,B 0,C 180,E1 8209.224,E2 8209.224} C_VEL
LIN {X 0,Y 449.868,Z 564.491,A -85,B 0,C 180,E1 8213.158,E2 8213.158} C_VEL
LIN {X 0,Y 453.028,Z 533.737,A -85,B 0,C 180,E1 8216.546,E2 8216.546} C_VEL
LIN {X 0,Y 456.501,Z 498.891,A -85,B 0,C 180,E1 8219.345,E2 8219.345} C_VEL
LIN {X 0,Y 459.684,Z 462.23,A -85,B 0,C 180,E1 8221.342,E2 8221.342} C_VEL
LIN {X 0,Y 461.867,Z 426.564,A -85,B 0,C 180,E1 8222.546,E2 8222.546} C_VEL
LIN {X 0,Y 461.58,Z 416.553,A -85,B 0,C 180,E1 8222.815,E2 8222.815} C_VEL
LIN {X 0,Y 444.715,Z 374.969,A -85,B 0,C 180,E1 8224.916,E2 8224.916} C_VEL
LIN {X 0,Y 443.063,Z 370.16,A -85,B 0,C 180,E1 8225.248,E2 8225.248} C_VEL
LIN {X 0,Y 442.773,Z 370.16,A -85,B 0,C 180,E1 8231.216,E2 8231.216} C_VEL
LIN {X 0,Y 442.685,Z 370.16,A -85,B 0,C 180,E1 8236.844,E2 8236.844} C_VEL
LIN {X 0,Y 442.814,Z 370.16,A -85,B 0,C 180,E1 8242.018,E2 8242.018} C_VEL
LIN {X 0,Y 442.945,Z 370.16,A -85,B 0,C 180,E1 8248.695,E2 8248.695} C_VEL
LIN {X 0,Y 443.186,Z 370.754,A -85,B 0,C 180,E1 8252.189,E2 8252.189} C_VEL
LIN {X 0,Y 454.129,Z 403.189,A -85,B 0,C 180,E1 8253.712,E2 8253.712} C_VEL
LIN {X 0,Y 455.089,Z 416.985,A -85,B 0,C 180,E1 8254.24,E2 8254.24} C_VEL
LIN {X 0,Y 453.42,Z 450.747,A -85,B 0,C 180,E1 8255.856,E2 8255.856} C_VEL
LIN {X 0,Y 451.365,Z 481.881,A -85,B 0,C 180,E1 8258.178,E2 8258.178} C_VEL
LIN {X 0,Y 449.06,Z 509.199,A -85,B 0,C 180,E1 8261.132,E2 8261.132} C_VEL
LIN {X 0,Y 447.267,Z 531.458,A -85,B 0,C 180,E1 8264.549,E2 8264.549} C_VEL
LIN {X 0,Y 445.874,Z 548.304,A -85,B 0,C 180,E1 8268.244,E2 8268.244} C_VEL
LIN {X 0,Y 445.064,Z 560.088,A -85,B 0,C 180,E1 8272.179,E2 8272.179} C_VEL
LIN {X 0,Y 444.721,Z 566.676,A -85,B 0,C 180,E1 8276.095,E2 8276.095} C_VEL
LIN {X 0,Y 444.571,Z 568.625,A -85,B 0,C 180,E1 8279.999,E2 8279.999} C_VEL
LIN {X 0,Y 444.633,Z 565.973,A -85,B 0,C 180,E1 8283.903,E2 8283.903} C_VEL
LIN {X 0,Y 444.964,Z 558.705,A -85,B 0,C 180,E1 8287.82,E2 8287.82} C_VEL
LIN {X 0,Y 445.696,Z 546.219,A -85,B 0,C 180,E1 8291.758,E2 8291.758} C_VEL
LIN {X 0,Y 447.12,Z 527.324,A -85,B 0,C 180,E1 8295.715,E2 8295.715} C_VEL
LIN {X 0,Y 448.91,Z 504.438,A -85,B 0,C 180,E1 8299.078,E2 8299.078} C_VEL
LIN {X 0,Y 451.269,Z 476.647,A -85,B 0,C 180,E1 8301.986,E2 8301.986} C_VEL
LIN {X 0,Y 453.429,Z 445.31,A -85,B 0,C 180,E1 8304.272,E2 8304.272} C_VEL
LIN {X 0,Y 455.183,Z 412.027,A -85,B 0,C 180,E1 8305.837,E2 8305.837} C_VEL
LIN {X 0,Y 449.6,Z 389.801,A -85,B 0,C 180,E1 8306.794,E2 8306.794} C_VEL
LIN {X 0,Y 443.178,Z 370.16,A -85,B 0,C 180,E1 8307.615,E2 8307.615} C_VEL
LIN {X 0,Y 443.027,Z 370.16,A -85,B 0,C 180,E1 8314.907,E2 8314.907} C_VEL
LIN {X 0,Y 442.9,Z 370.16,A -85,B 0,C 180,E1 8321.24,E2 8321.24} C_VEL
LIN {X 0,Y 442.89,Z 370.16,A -85,B 0,C 180,E1 8326.874,E2 8326.874} C_VEL
LIN {X 0,Y 442.897,Z 370.16,A -85,B 0,C 180,E1 8332.031,E2 8332.031} C_VEL
LIN {X 0,Y 442.949,Z 370.16,A -85,B 0,C 180,E1 8338.696,E2 8338.696} C_VEL
LIN {X 0,Y 443.098,Z 370.16,A -85,B 0,C 180,E1 8339.972,E2 8339.972} C_VEL
LIN {X 0,Y 459.89,Z 410.854,A -85,B 0,C 180,E1 8342.331,E2 8342.331} C_VEL
LIN {X 0,Y 461.184,Z 417.454,A -85,B 0,C 180,E1 8342.694,E2 8342.694} C_VEL
LIN {X 0,Y 458.649,Z 449.668,A -85,B 0,C 180,E1 8344.31,E2 8344.31} C_VEL
LIN {X 0,Y 455.394,Z 479.626,A -85,B 0,C 180,E1 8346.621,E2 8346.621} C_VEL
LIN {X 0,Y 451.876,Z 506.622,A -85,B 0,C 180,E1 8349.645,E2 8349.645} C_VEL
LIN {X 0,Y 448.89,Z 528.544,A -85,B 0,C 180,E1 8353.092,E2 8353.092} C_VEL
LIN {X 0,Y 446.755,Z 545.157,A -85,B 0,C 180,E1 8356.78,E2 8356.78} C_VEL
LIN {X 0,Y 445.316,Z 558.532,A -85,B 0,C 180,E1 8361.203,E2 8361.203} C_VEL
LIN {X 0,Y 444.663,Z 566.554,A -85,B 0,C 180,E1 8366.098,E2 8366.098} C_VEL
LIN {X 0,Y 444.526,Z 568.427,A -85,B 0,C 180,E1 8370.003,E2 8370.003} C_VEL
LIN {X 0,Y 444.786,Z 565.326,A -85,B 0,C 180,E1 8374.884,E2 8374.884} C_VEL
LIN {X 0,Y 445.485,Z 556.491,A -85,B 0,C 180,E1 8379.527,E2 8379.527} C_VEL
LIN {X 0,Y 447.007,Z 542.91,A -85,B 0,C 180,E1 8383.717,E2 8383.717} C_VEL
LIN {X 0,Y 449.531,Z 523.873,A -85,B 0,C 180,E1 8387.647,E2 8387.647} C_VEL
LIN {X 0,Y 452.628,Z 501.142,A -85,B 0,C 180,E1 8390.966,E2 8390.966} C_VEL
LIN {X 0,Y 456.079,Z 473.758,A -85,B 0,C 180,E1 8393.81,E2 8393.81} C_VEL
LIN {X 0,Y 459.227,Z 442.921,A -85,B 0,C 180,E1 8396.002,E2 8396.002} C_VEL
LIN {X 0,Y 460.751,Z 413.247,A -85,B 0,C 180,E1 8397.413,E2 8397.413} C_VEL
LIN {X 0,Y 446.859,Z 379.491,A -85,B 0,C 180,E1 8399.417,E2 8399.417} C_VEL
LIN {X 0,Y 443.028,Z 370.16,A -85,B 0,C 180,E1 8399.947,E2 8399.947} C_VEL
LIN {X 0,Y 442.876,Z 370.16,A -85,B 0,C 180,E1 8405.534,E2 8405.534} C_VEL
LIN {X 0,Y 442.774,Z 370.16,A -85,B 0,C 180,E1 8411.22,E2 8411.22} C_VEL
LIN {X 0,Y 442.847,Z 370.16,A -85,B 0,C 180,E1 8416.867,E2 8416.867} C_VEL
LIN {X 0,Y 442.868,Z 370.16,A -85,B 0,C 180,E1 8422.027,E2 8422.027} C_VEL
LIN {X 0,Y 442.901,Z 370.16,A -85,B 0,C 180,E1 8428.716,E2 8428.716} C_VEL
LIN {X 0,Y 443.129,Z 370.16,A -85,B 0,C 180,E1 8433.634,E2 8433.634} C_VEL
LIN {X 0,Y 443.356,Z 370.16,A -85,B 0,C 180,E1 8440.035,E2 8440.035} C_VEL
LIN {X 0,Y 443.562,Z 370.16,A -85,B 0,C 180,E1 8446.179,E2 8446.179} C_VEL
LIN {X 0,Y 443.691,Z 370.16,A -85,B 0,C 180,E1 8452.157,E2 8452.157} C_VEL
LIN {X 0,Y 443.878,Z 370.16,A -85,B 0,C 180,E1 8458.047,E2 8458.047} C_VEL
LIN {X 0,Y 443.787,Z 370.16,A -85,B 0,C 180,E1 8463.913,E2 8463.913} C_VEL
LIN {X 0,Y 443.611,Z 370.16,A -85,B 0,C 180,E1 8469.826,E2 8469.826} C_VEL
LIN {X 0,Y 443.402,Z 370.16,A -85,B 0,C 180,E1 8475.853,E2 8475.853} C_VEL
LIN {X 0,Y 443.247,Z 370.16,A -85,B 0,C 180,E1 8482.069,E2 8482.069} C_VEL
LIN {X 0,Y 443.032,Z 370.16,A -85,B 0,C 180,E1 8488.582,E2 8488.582} C_VEL
LIN {X 0,Y 442.993,Z 370.16,A -85,B 0,C 180,E1 8495.52,E2 8495.52} C_VEL
LIN {X 0,Y 442.869,Z 370.16,A -85,B 0,C 180,E1 8501.226,E2 8501.226} C_VEL
LIN {X 0,Y 442.866,Z 370.16,A -85,B 0,C 180,E1 8506.863,E2 8506.863} C_VEL
LIN {X 0,Y 442.9,Z 370.16,A -85,B 0,C 180,E1 8512.024,E2 8512.024} C_VEL
LIN {X 0,Y 442.953,Z 370.16,A -85,B 0,C 180,E1 8514.826,E2 8514.826} C_VEL
LIN {X 0,Y 461.908,Z 417.554,A -85,B 0,C 180,E1 8517.232,E2 8517.232} C_VEL
LIN {X 0,Y 459.968,Z 457.106,A -85,B 0,C 180,E1 8518.432,E2 8518.432} C_VEL
LIN {X 0,Y 457.047,Z 493.283,A -85,B 0,C 180,E1 8520.302,E2 8520.302} C_VEL
LIN {X 0,Y 456.41,Z 500.677,A -85,B 0,C 180,E1 8520.784,E2 8520.784} C_VEL
LIN {X 0,Y 453.012,Z 512.157,A -85,B 0,C 180,E1 8521.491,E2 8521.491} C_VEL
LIN {X 0,Y 446.242,Z 528.539,A -85,B 0,C 180,E1 8522.598,E2 8522.598} C_VEL
LIN {X 0,Y 445.986,Z 530.285,A -85,B 0,C 180,E1 8522.762,E2 8522.762} C_VEL
LIN {X 0,Y 442.55,Z 561.241,A -85,B 0,C 180,E1 8526.162,E2 8526.162} C_VEL
LIN {X 0,Y 439.7,Z 588.418,A -85,B 0,C 180,E1 8530.205,E2 8530.205} C_VEL
LIN {X 0,Y 437.856,Z 609.065,A -85,B 0,C 180,E1 8534.421,E2 8534.421} C_VEL
LIN {X 0,Y 436.838,Z 624.808,A -85,B 0,C 180,E1 8539.009,E2 8539.009} C_VEL
LIN {X 0,Y 436.543,Z 633.752,A -85,B 0,C 180,E1 8543.025,E2 8543.025} C_VEL
LIN {X 0,Y 436.397,Z 637.733,A -85,B 0,C 180,E1 8546.018,E2 8546.018} C_VEL
LIN {X 0,Y 436.382,Z 639.702,A -85,B 0,C 180,E1 8549.997,E2 8549.997} C_VEL
LIN {X 0,Y 436.453,Z 636.666,A -85,B 0,C 180,E1 8554.972,E2 8554.972} C_VEL
LIN {X 0,Y 436.666,Z 629.345,A -85,B 0,C 180,E1 8559.2,E2 8559.2} C_VEL
LIN {X 0,Y 437.332,Z 616.97,A -85,B 0,C 180,E1 8563.51,E2 8563.51} C_VEL
LIN {X 0,Y 438.64,Z 598.839,A -85,B 0,C 180,E1 8567.834,E2 8567.834} C_VEL
LIN {X 0,Y 440.98,Z 575.102,A -85,B 0,C 180,E1 8571.93,E2 8571.93} C_VEL
LIN {X 0,Y 444.248,Z 546.314,A -85,B 0,C 180,E1 8575.613,E2 8575.613} C_VEL
LIN {X 0,Y 447.858,Z 513.389,A -85,B 0,C 180,E1 8578.689,E2 8578.689} C_VEL
LIN {X 0,Y 451.353,Z 477.821,A -85,B 0,C 180,E1 8581.046,E2 8581.046} C_VEL
LIN {X 0,Y 454.156,Z 440.591,A -85,B 0,C 180,E1 8582.635,E2 8582.635} C_VEL
LIN {X 0,Y 454.81,Z 419.048,A -85,B 0,C 180,E1 8583.244,E2 8583.244} C_VEL
LIN {X 0,Y 438.811,Z 379.358,A -85,B 0,C 180,E1 8585.309,E2 8585.309} C_VEL
LIN {X 0,Y 435.085,Z 370.16,A -85,B 0,C 180,E1 8585.851,E2 8585.851} C_VEL
LIN {X 0,Y 434.808,Z 370.16,A -85,B 0,C 180,E1 8593.013,E2 8593.013} C_VEL
LIN {X 0,Y 434.797,Z 370.16,A -85,B 0,C 180,E1 8599.993,E2 8599.993} C_VEL
LIN {X 0,Y 435.022,Z 370.16,A -85,B 0,C 180,E1 8606.634,E2 8606.634} C_VEL
LIN {X 0,Y 435.179,Z 370.16,A -85,B 0,C 180,E1 8611.517,E2 8611.517} C_VEL
LIN {X 0,Y 446.762,Z 403.65,A -85,B 0,C 180,E1 8613.238,E2 8613.238} C_VEL
LIN {X 0,Y 448.002,Z 416.237,A -85,B 0,C 180,E1 8613.756,E2 8613.756} C_VEL
LIN {X 0,Y 446.297,Z 450.112,A -85,B 0,C 180,E1 8615.375,E2 8615.375} C_VEL
LIN {X 0,Y 444.168,Z 480.783,A -85,B 0,C 180,E1 8617.65,E2 8617.65} C_VEL
LIN {X 0,Y 441.819,Z 507.471,A -85,B 0,C 180,E1 8620.488,E2 8620.488} C_VEL
LIN {X 0,Y 439.81,Z 530.742,A -85,B 0,C 180,E1 8624.014,E2 8624.014} C_VEL
LIN {X 0,Y 438.299,Z 547.105,A -85,B 0,C 180,E1 8627.532,E2 8627.532} C_VEL
LIN {X 0,Y 437.421,Z 558.873,A -85,B 0,C 180,E1 8631.229,E2 8631.229} C_VEL
LIN {X 0,Y 436.926,Z 566.228,A -85,B 0,C 180,E1 8635.029,E2 8635.029} C_VEL
LIN {X 0,Y 436.805,Z 568.878,A -85,B 0,C 180,E1 8638.013,E2 8638.013} C_VEL
LIN {X 0,Y 436.611,Z 568.494,A -85,B 0,C 180,E1 8641.986,E2 8641.986} C_VEL
LIN {X 0,Y 436.94,Z 562.534,A -85,B 0,C 180,E1 8646.464,E2 8646.464} C_VEL
LIN {X 0,Y 437.491,Z 552.025,A -85,B 0,C 180,E1 8650.466,E2 8650.466} C_VEL
LIN {X 0,Y 438.734,Z 535.292,A -85,B 0,C 180,E1 8654.532,E2 8654.532} C_VEL
LIN {X 0,Y 440.614,Z 513.498,A -85,B 0,C 180,E1 8658.191,E2 8658.191} C_VEL
LIN {X 0,Y 442.95,Z 486.313,A -85,B 0,C 180,E1 8661.423,E2 8661.423} C_VEL
LIN {X 0,Y 445.366,Z 456.352,A -85,B 0,C 180,E1 8663.92,E2 8663.92} C_VEL
LIN {X 0,Y 447.289,Z 423.865,A -85,B 0,C 180,E1 8665.741,E2 8665.741} C_VEL
LIN {X 0,Y 447.141,Z 407.794,A -85,B 0,C 180,E1 8666.398,E2 8666.398} C_VEL
LIN {X 0,Y 435.218,Z 370.16,A -85,B 0,C 180,E1 8668.047,E2 8668.047} C_VEL
LIN {X 0,Y 435.06,Z 370.16,A -85,B 0,C 180,E1 8673.831,E2 8673.831} C_VEL
LIN {X 0,Y 434.979,Z 370.16,A -85,B 0,C 180,E1 8680.035,E2 8680.035} C_VEL
LIN {X 0,Y 435.013,Z 370.16,A -85,B 0,C 180,E1 8685.894,E2 8685.894} C_VEL
LIN {X 0,Y 434.924,Z 370.16,A -85,B 0,C 180,E1 8691.207,E2 8691.207} C_VEL
LIN {X 0,Y 435.044,Z 370.16,A -85,B 0,C 180,E1 8698.538,E2 8698.538} C_VEL
LIN {X 0,Y 435.111,Z 370.16,A -85,B 0,C 180,E1 8699.319,E2 8699.319} C_VEL
LIN {X 0,Y 451.824,Z 409.893,A -85,B 0,C 180,E1 8701.682,E2 8701.682} C_VEL
LIN {X 0,Y 454.31,Z 418.984,A -85,B 0,C 180,E1 8702.245,E2 8702.245} C_VEL
LIN {X 0,Y 451.614,Z 450.728,A -85,B 0,C 180,E1 8703.88,E2 8703.88} C_VEL
LIN {X 0,Y 448.2,Z 480.528,A -85,B 0,C 180,E1 8706.223,E2 8706.223} C_VEL
LIN {X 0,Y 444.513,Z 507.199,A -85,B 0,C 180,E1 8709.262,E2 8709.262} C_VEL
LIN {X 0,Y 441.32,Z 529.269,A -85,B 0,C 180,E1 8712.793,E2 8712.793} C_VEL
LIN {X 0,Y 439.034,Z 545.85,A -85,B 0,C 180,E1 8716.543,E2 8716.543} C_VEL
LIN {X 0,Y 437.594,Z 558.164,A -85,B 0,C 180,E1 8720.612,E2 8720.612} C_VEL
LIN {X 0,Y 436.926,Z 566.083,A -85,B 0,C 180,E1 8725.034,E2 8725.034} C_VEL
LIN {X 0,Y 436.664,Z 569.063,A -85,B 0,C 180,E1 8730.003,E2 8730.003} C_VEL
LIN {X 0,Y 436.944,Z 565.97,A -85,B 0,C 180,E1 8734.972,E2 8734.972} C_VEL
LIN {X 0,Y 437.625,Z 557.917,A -85,B 0,C 180,E1 8739.395,E2 8739.395} C_VEL
LIN {X 0,Y 439.083,Z 545.489,A -85,B 0,C 180,E1 8743.461,E2 8743.461} C_VEL
LIN {X 0,Y 441.611,Z 527.391,A -85,B 0,C 180,E1 8747.459,E2 8747.459} C_VEL
LIN {X 0,Y 445.049,Z 503.713,A -85,B 0,C 180,E1 8751.109,E2 8751.109} C_VEL
LIN {X 0,Y 448.727,Z 476.075,A -85,B 0,C 180,E1 8754.087,E2 8754.087} C_VEL
LIN {X 0,Y 452.102,Z 445.51,A -85,B 0,C 180,E1 8756.353,E2 8756.353} C_VEL
LIN {X 0,Y 453.726,Z 415.397,A -85,B 0,C 180,E1 8757.851,E2 8757.851} C_VEL
LIN {X 0,Y 440.691,Z 383.219,A -85,B 0,C 180,E1 8759.856,E2 8759.856} C_VEL
LIN {X 0,Y 435.075,Z 370.16,A -85,B 0,C 180,E1 8760.575,E2 8760.575} C_VEL
LIN {X 0,Y 434.85,Z 370.16,A -85,B 0,C 180,E1 8766.802,E2 8766.802} C_VEL
LIN {X 0,Y 434.873,Z 370.16,A -85,B 0,C 180,E1 8773.026,E2 8773.026} C_VEL
LIN {X 0,Y 434.946,Z 370.16,A -85,B 0,C 180,E1 8778.601,E2 8778.601} C_VEL
LIN {X 0,Y 434.892,Z 370.16,A -85,B 0,C 180,E1 8783.718,E2 8783.718} C_VEL
LIN {X 0,Y 435.012,Z 370.16,A -85,B 0,C 180,E1 8790.471,E2 8790.471} C_VEL
LIN {X 0,Y 435.242,Z 370.16,A -85,B 0,C 180,E1 8795.331,E2 8795.331} C_VEL
LIN {X 0,Y 435.464,Z 370.16,A -85,B 0,C 180,E1 8801.768,E2 8801.768} C_VEL
LIN {X 0,Y 435.669,Z 370.16,A -85,B 0,C 180,E1 8807.967,E2 8807.967} C_VEL
LIN {X 0,Y 435.821,Z 370.16,A -85,B 0,C 180,E1 8814.02,E2 8814.02} C_VEL
LIN {X 0,Y 436.127,Z 370.16,A -85,B 0,C 180,E1 8820.001,E2 8820.001} C_VEL
LIN {X 0,Y 435.884,Z 370.16,A -85,B 0,C 180,E1 8825.982,E2 8825.982} C_VEL
LIN {X 0,Y 435.583,Z 370.16,A -85,B 0,C 180,E1 8832.038,E2 8832.038} C_VEL
LIN {X 0,Y 435.432,Z 370.16,A -85,B 0,C 180,E1 8838.236,E2 8838.236} C_VEL
LIN {X 0,Y 435.24,Z 370.16,A -85,B 0,C 180,E1 8844.672,E2 8844.672} C_VEL
LIN {X 0,Y 435.034,Z 370.16,A -85,B 0,C 180,E1 8851.468,E2 8851.468} C_VEL
LIN {X 0,Y 434.962,Z 370.16,A -85,B 0,C 180,E1 8856.814,E2 8856.814} C_VEL
LIN {X 0,Y 434.946,Z 370.16,A -85,B 0,C 180,E1 8863.029,E2 8863.029} C_VEL
LIN {X 0,Y 434.965,Z 370.16,A -85,B 0,C 180,E1 8868.596,E2 8868.596} C_VEL
LIN {X 0,Y 435.019,Z 370.773,A -85,B 0,C 180,E1 8874.199,E2 8874.199} C_VEL
LIN {X 0,Y 453.117,Z 414.808,A -85,B 0,C 180,E1 8876.538,E2 8876.538} C_VEL
LIN {X 0,Y 455.187,Z 422.516,A -85,B 0,C 180,E1 8876.868,E2 8876.868} C_VEL
LIN {X 0,Y 452.799,Z 459.824,A -85,B 0,C 180,E1 8878.089,E2 8878.089} C_VEL
LIN {X 0,Y 449.748,Z 494.467,A -85,B 0,C 180,E1 8879.949,E2 8879.949} C_VEL
LIN {X 0,Y 446.164,Z 528.566,A -85,B 0,C 180,E1 8882.596,E2 8882.596} C_VEL
LIN {X 0,Y 445.986,Z 530.285,A -85,B 0,C 180,E1 8882.762,E2 8882.762} C_VEL
LIN {X 0,Y 442.503,Z 540.813,A -85,B 0,C 180,E1 8883.69,E2 8883.69} C_VEL
LIN {X 0,Y 435.682,Z 555.675,A -85,B 0,C 180,E1 8885.141,E2 8885.141} C_VEL
LIN {X 0,Y 435.416,Z 557.233,A -85,B 0,C 180,E1 8885.338,E2 8885.338} C_VEL
LIN {X 0,Y 432.397,Z 584.075,A -85,B 0,C 180,E1 8889.264,E2 8889.264} C_VEL
LIN {X 0,Y 430.24,Z 606.182,A -85,B 0,C 180,E1 8893.647,E2 8893.647} C_VEL
LIN {X 0,Y 429.067,Z 622.6,A -85,B 0,C 180,E1 8898.291,E2 8898.291} C_VEL
LIN {X 0,Y 428.673,Z 633.061,A -85,B 0,C 180,E1 8902.897,E2 8902.897} C_VEL
LIN {X 0,Y 428.52,Z 637.079,A -85,B 0,C 180,E1 8905.945,E2 8905.945} C_VEL
LIN {X 0,Y 428.507,Z 639.065,A -85,B 0,C 180,E1 8909.997,E2 8909.997} C_VEL
LIN {X 0,Y 428.562,Z 635.996,A -85,B 0,C 180,E1 8915.064,E2 8915.064} C_VEL
LIN {X 0,Y 428.821,Z 627.762,A -85,B 0,C 180,E1 8919.721,E2 8919.721} C_VEL
LIN {X 0,Y 429.597,Z 614.261,A -85,B 0,C 180,E1 8924.278,E2 8924.278} C_VEL
LIN {X 0,Y 431.114,Z 596.057,A -85,B 0,C 180,E1 8928.53,E2 8928.53} C_VEL
LIN {X 0,Y 433.81,Z 570.727,A -85,B 0,C 180,E1 8932.842,E2 8932.842} C_VEL
LIN {X 0,Y 437.152,Z 542.652,A -85,B 0,C 180,E1 8936.361,E2 8936.361} C_VEL
LIN {X 0,Y 440.868,Z 511.056,A -85,B 0,C 180,E1 8939.294,E2 8939.294} C_VEL
LIN {X 0,Y 444.543,Z 475.435,A -85,B 0,C 180,E1 8941.635,E2 8941.635} C_VEL
LIN {X 0,Y 447.374,Z 439.413,A -85,B 0,C 180,E1 8943.164,E2 8943.164} C_VEL
LIN {X 0,Y 447.939,Z 421.292,A -85,B 0,C 180,E1 8943.703,E2 8943.703} C_VEL
LIN {X 0,Y 432.82,Z 383.52,A -85,B 0,C 180,E1 8945.727,E2 8945.727} C_VEL
LIN {X 0,Y 427.1,Z 370.16,A -85,B 0,C 180,E1 8946.63,E2 8946.63} C_VEL
LIN {X 0,Y 426.898,Z 370.16,A -85,B 0,C 180,E1 8952.357,E2 8952.357} C_VEL
LIN {X 0,Y 426.872,Z 370.16,A -85,B 0,C 180,E1 8958.136,E2 8958.136} C_VEL
LIN {X 0,Y 426.928,Z 370.16,A -85,B 0,C 180,E1 8964.642,E2 8964.642} C_VEL
LIN {X 0,Y 427.194,Z 370.269,A -85,B 0,C 180,E1 8970.845,E2 8970.845} C_VEL
LIN {X 0,Y 439.166,Z 402.896,A -85,B 0,C 180,E1 8972.676,E2 8972.676} C_VEL
LIN {X 0,Y 441.021,Z 416.154,A -85,B 0,C 180,E1 8973.274,E2 8973.274} C_VEL
